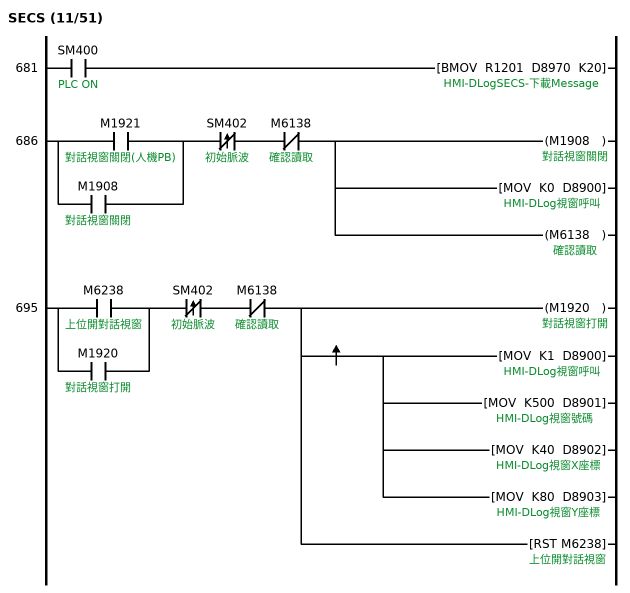
681   LD      SM400  ; PLC ON
      BMOV    R1201 D8970 K20  ; HMI-DLogSECS-下載Message
686   LD      M1921  ; 對話視窗關閉(人機PB)
      OR      M1908  ; 對話視窗關閉
      ANDPI   SM402  ; 初始脈波
      ANI     M6138  ; 確認讀取
      OUT     M1908  ; 對話視窗關閉
      MOV     K0 D8900  ; HMI-DLog視窗呼叫
      OUT     M6138  ; 確認讀取
695   LD      M6238  ; 上位開對話視窗
      OR      M1920  ; 對話視窗打開
      ANDPI   SM402  ; 初始脈波
      ANI     M6138  ; 確認讀取
      OUT     M1920  ; 對話視窗打開
      MPS
      MEP
      MOV     K1 D8900
      MOV     K500 D8901  ; HMI-DLog視窗號碼
      MOV     K40 D8902  ; HMI-DLog視窗X座標
      MOV     K80 D8903  ; HMI-DLog視窗Y座標
      MPP
      RST     M6238  ; 上位開對話視窗
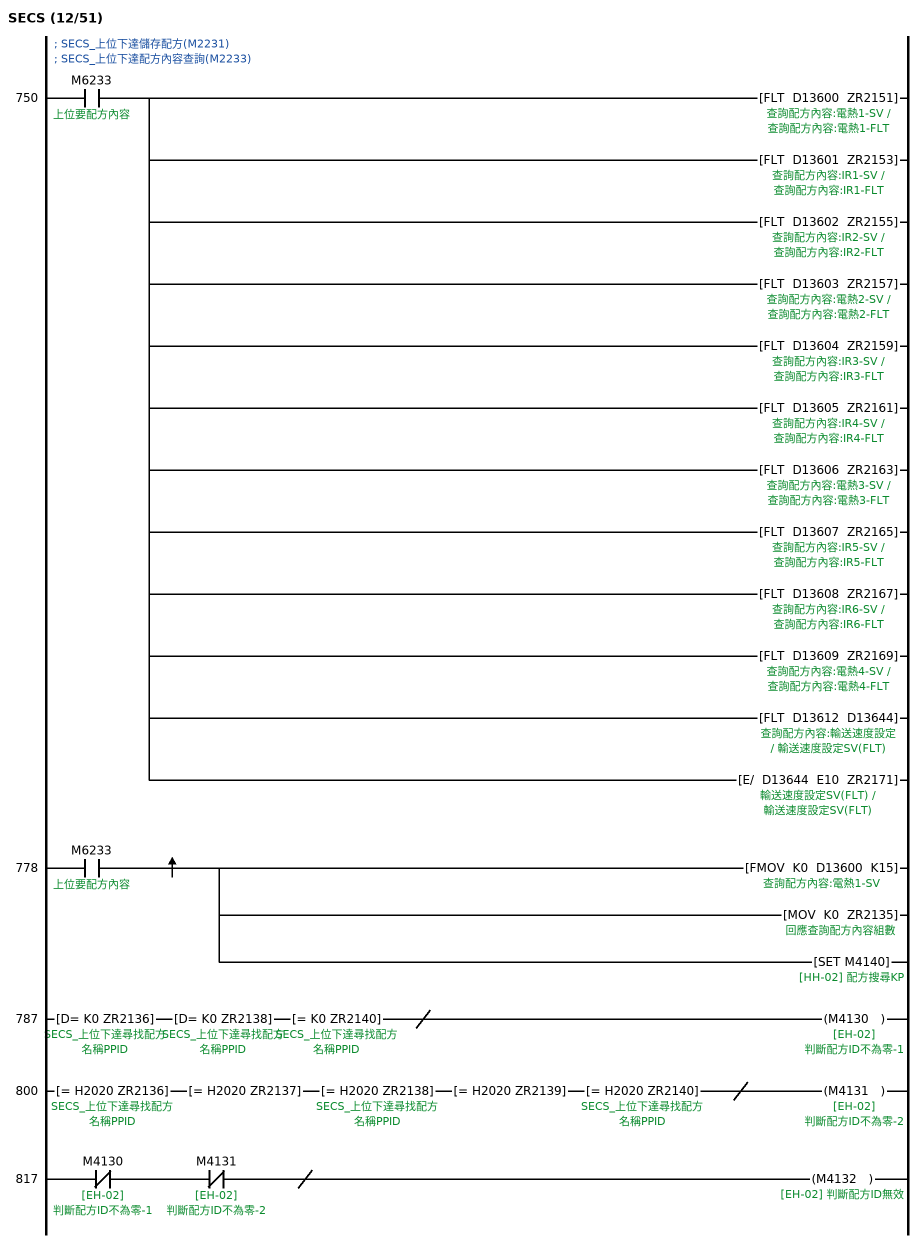
; SECS_上位下達儲存配方(M2231)
; SECS_上位下達配方內容查詢(M2233)
750   LD      M6233  ; 上位要配方內容
      FLT     D13600 ZR2151  ; 查詢配方內容:電熱1-SV / 查詢配方內容:電熱1-FLT
      FLT     D13601 ZR2153  ; 查詢配方內容:IR1-SV / 查詢配方內容:IR1-FLT
      FLT     D13602 ZR2155  ; 查詢配方內容:IR2-SV / 查詢配方內容:IR2-FLT
      FLT     D13603 ZR2157  ; 查詢配方內容:電熱2-SV / 查詢配方內容:電熱2-FLT
      FLT     D13604 ZR2159  ; 查詢配方內容:IR3-SV / 查詢配方內容:IR3-FLT
      FLT     D13605 ZR2161  ; 查詢配方內容:IR4-SV / 查詢配方內容:IR4-FLT
      FLT     D13606 ZR2163  ; 查詢配方內容:電熱3-SV / 查詢配方內容:電熱3-FLT
      FLT     D13607 ZR2165  ; 查詢配方內容:IR5-SV / 查詢配方內容:IR5-FLT
      FLT     D13608 ZR2167  ; 查詢配方內容:IR6-SV / 查詢配方內容:IR6-FLT
      FLT     D13609 ZR2169  ; 查詢配方內容:電熱4-SV / 查詢配方內容:電熱4-FLT
      FLT     D13612 D13644  ; 查詢配方內容:輸送速度設定 / 輸送速度設定SV(FLT)
      E/      D13644 E10 ZR2171  ; 輸送速度設定SV(FLT)
778   LD      M6233  ; 上位要配方內容
      MEP
      FMOV    K0 D13600 K15
      MOV     K0 ZR2135  ; 回應查詢配方內容組數
      SET     M4140  ; [HH-02] 配方搜尋KP
787   LDD=    K0 ZR2136  ; SECS_上位下達尋找配方名稱PPID
      ANDD=   K0 ZR2138  ; SECS_上位下達尋找配方名稱PPID
      AND=    K0 ZR2140  ; SECS_上位下達尋找配方名稱PPID
      INV
      OUT     M4130  ; [EH-02] 判斷配方ID不為零-1
800   LD=     H2020 ZR2136  ; SECS_上位下達尋找配方名稱PPID
      AND=    H2020 ZR2137
      AND=    H2020 ZR2138  ; SECS_上位下達尋找配方名稱PPID
      AND=    H2020 ZR2139
      AND=    H2020 ZR2140  ; SECS_上位下達尋找配方名稱PPID
      INV
      OUT     M4131  ; [EH-02] 判斷配方ID不為零-2
817   LDI     M4130  ; [EH-02] 判斷配方ID不為零-1
      ANI     M4131  ; [EH-02] 判斷配方ID不為零-2
      INV
      OUT     M4132  ; [EH-02] 判斷配方ID無效
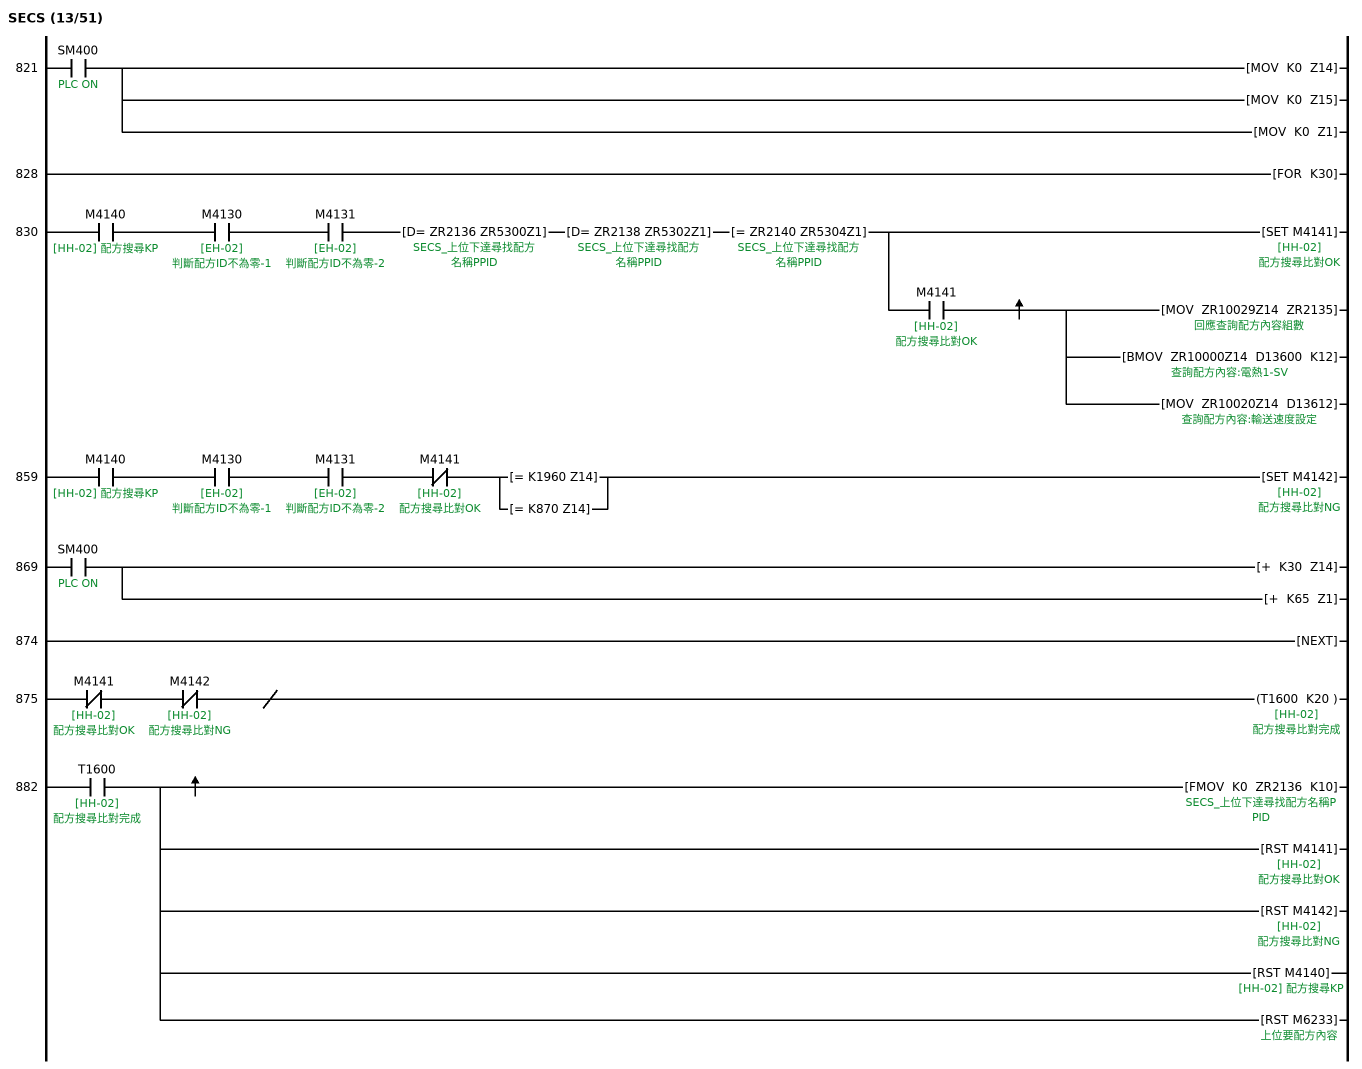
821   LD      SM400  ; PLC ON
      MOV     K0 Z14
      MOV     K0 Z15
      MOV     K0 Z1
828   FOR     K30
830   LD      M4140  ; [HH-02] 配方搜尋KP
      AND     M4130  ; [EH-02] 判斷配方ID不為零-1
      AND     M4131  ; [EH-02] 判斷配方ID不為零-2
      ANDD=   ZR2136 ZR5300Z1  ; SECS_上位下達尋找配方名稱PPID
      ANDD=   ZR2138 ZR5302Z1  ; SECS_上位下達尋找配方名稱PPID
      AND=    ZR2140 ZR5304Z1  ; SECS_上位下達尋找配方名稱PPID
      SET     M4141  ; [HH-02] 配方搜尋比對OK
      AND     M4141  ; [HH-02] 配方搜尋比對OK
      MEP
      MOV     ZR10029Z14 ZR2135
      BMOV    ZR10000Z14 D13600 K12
      MOV     ZR10020Z14 D13612
859   LD      M4140  ; [HH-02] 配方搜尋KP
      AND     M4130  ; [EH-02] 判斷配方ID不為零-1
      AND     M4131  ; [EH-02] 判斷配方ID不為零-2
      ANI     M4141  ; [HH-02] 配方搜尋比對OK
      LD=     K1960 Z14
      OR=     K870 Z14
      ANB
      SET     M4142  ; [HH-02] 配方搜尋比對NG
869   LD      SM400  ; PLC ON
      +       K30 Z14
      +       K65 Z1
874   NEXT
875   LDI     M4141  ; [HH-02] 配方搜尋比對OK
      ANI     M4142  ; [HH-02] 配方搜尋比對NG
      INV
      OUT     T1600 K20  ; [HH-02] 配方搜尋比對完成
882   LD      T1600  ; [HH-02] 配方搜尋比對完成
      MPS
      MEP
      FMOV    K0 ZR2136 K10
      MPP
      RST     M4141  ; [HH-02] 配方搜尋比對OK
      RST     M4142  ; [HH-02] 配方搜尋比對NG
      RST     M4140  ; [HH-02] 配方搜尋KP
      RST     M6233  ; 上位要配方內容
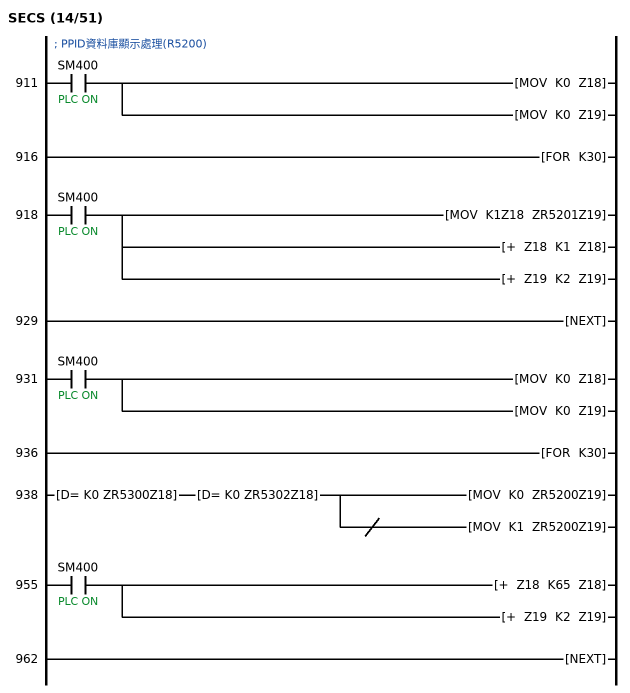
; PPID資料庫顯示處理(R5200)
911   LD      SM400  ; PLC ON
      MOV     K0 Z18
      MOV     K0 Z19
916   FOR     K30
918   LD      SM400  ; PLC ON
      MOV     K1Z18 ZR5201Z19
      +       Z18 K1 Z18
      +       Z19 K2 Z19
929   NEXT
931   LD      SM400  ; PLC ON
      MOV     K0 Z18
      MOV     K0 Z19
936   FOR     K30
938   LDD=    K0 ZR5300Z18
      ANDD=   K0 ZR5302Z18
      MOV     K0 ZR5200Z19
      INV
      MOV     K1 ZR5200Z19
955   LD      SM400  ; PLC ON
      +       Z18 K65 Z18
      +       Z19 K2 Z19
962   NEXT
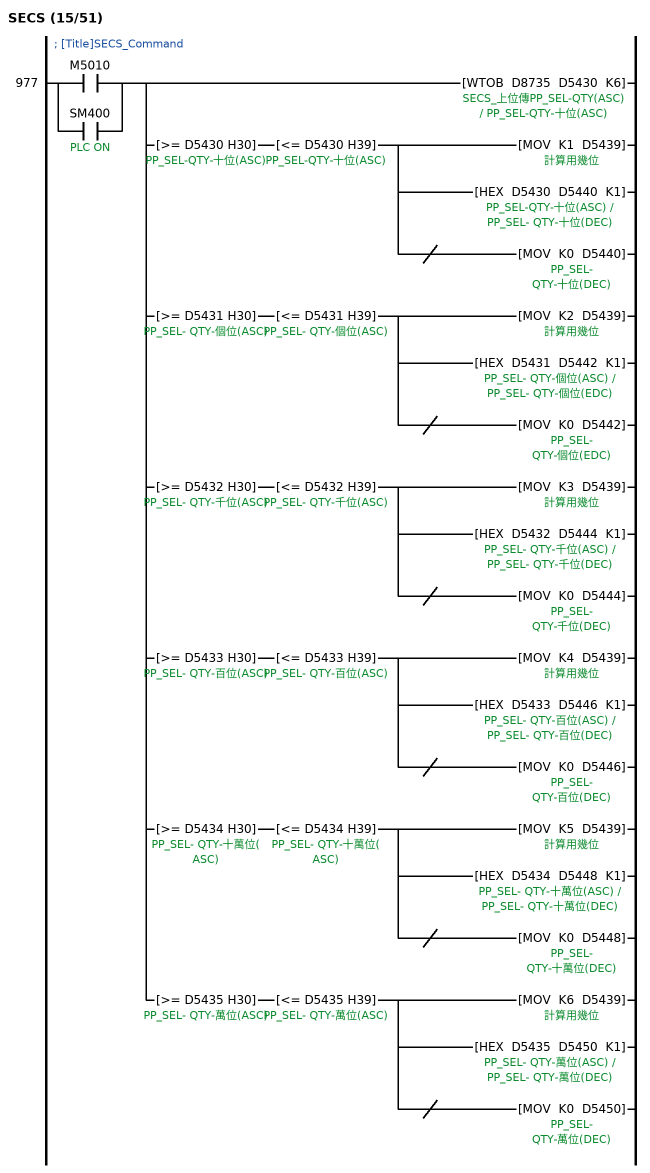
; [Title]SECS_Command
977   LD      M5010
      OR      SM400  ; PLC ON
      WTOB    D8735 D5430 K6  ; SECS_上位傳PP_SEL-QTY(ASC) / PP_SEL-QTY-十位(ASC)
      MPS
      AND>=   D5430 H30  ; PP_SEL-QTY-十位(ASC)
      AND<=   D5430 H39  ; PP_SEL-QTY-十位(ASC)
      MOV     K1 D5439  ; 計算用幾位
      HEX     D5430 D5440 K1  ; PP_SEL- QTY-十位(DEC)
      INV
      MOV     K0 D5440
      MRD
      AND>=   D5431 H30  ; PP_SEL- QTY-個位(ASC)
      AND<=   D5431 H39  ; PP_SEL- QTY-個位(ASC)
      MOV     K2 D5439
      HEX     D5431 D5442 K1  ; PP_SEL- QTY-個位(EDC)
      INV
      MOV     K0 D5442
      MRD
      AND>=   D5432 H30  ; PP_SEL- QTY-千位(ASC)
      AND<=   D5432 H39  ; PP_SEL- QTY-千位(ASC)
      MOV     K3 D5439
      HEX     D5432 D5444 K1  ; PP_SEL- QTY-千位(DEC)
      INV
      MOV     K0 D5444
      MRD
      AND>=   D5433 H30  ; PP_SEL- QTY-百位(ASC)
      AND<=   D5433 H39  ; PP_SEL- QTY-百位(ASC)
      MOV     K4 D5439
      HEX     D5433 D5446 K1  ; PP_SEL- QTY-百位(DEC)
      INV
      MOV     K0 D5446
      MRD
      AND>=   D5434 H30  ; PP_SEL- QTY-十萬位(ASC)
      AND<=   D5434 H39  ; PP_SEL- QTY-十萬位(ASC)
      MOV     K5 D5439
      HEX     D5434 D5448 K1  ; PP_SEL- QTY-十萬位(DEC)
      INV
      MOV     K0 D5448
      MPP
      AND>=   D5435 H30  ; PP_SEL- QTY-萬位(ASC)
      AND<=   D5435 H39  ; PP_SEL- QTY-萬位(ASC)
      MOV     K6 D5439
      HEX     D5435 D5450 K1  ; PP_SEL- QTY-萬位(DEC)
      INV
      MOV     K0 D5450
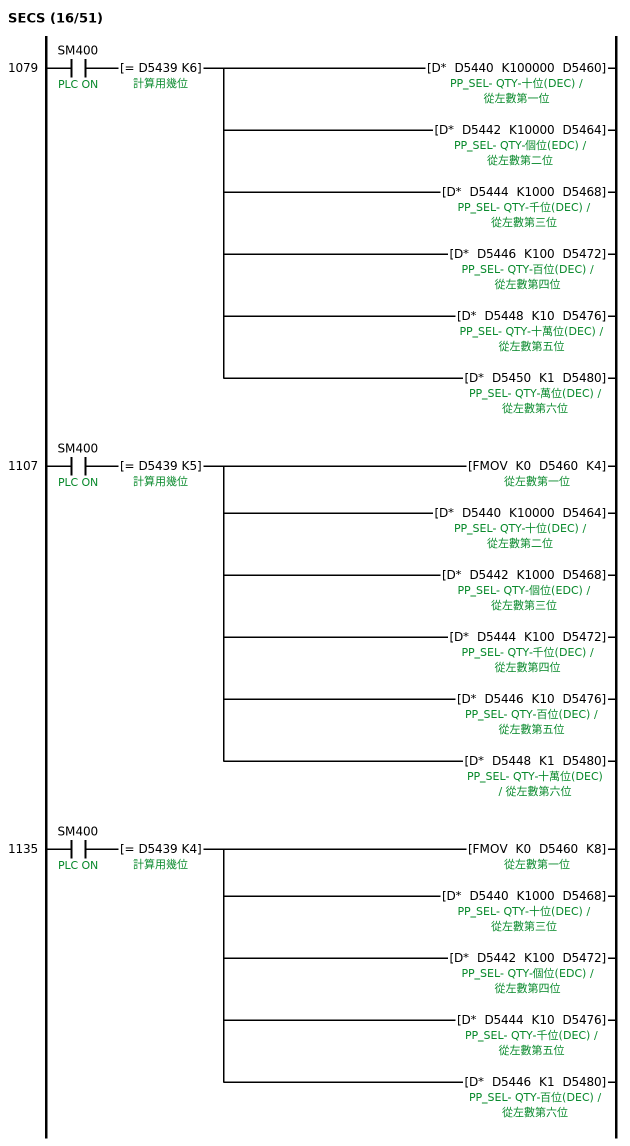
1079  LD      SM400  ; PLC ON
      AND=    D5439 K6  ; 計算用幾位
      D*      D5440 K100000 D5460  ; 從左數第一位
      D*      D5442 K10000 D5464  ; 從左數第二位
      D*      D5444 K1000 D5468  ; 從左數第三位
      D*      D5446 K100 D5472  ; 從左數第四位
      D*      D5448 K10 D5476  ; 從左數第五位
      D*      D5450 K1 D5480  ; 從左數第六位
1107  LD      SM400  ; PLC ON
      AND=    D5439 K5  ; 計算用幾位
      FMOV    K0 D5460 K4
      D*      D5440 K10000 D5464
      D*      D5442 K1000 D5468
      D*      D5444 K100 D5472
      D*      D5446 K10 D5476
      D*      D5448 K1 D5480
1135  LD      SM400  ; PLC ON
      AND=    D5439 K4  ; 計算用幾位
      FMOV    K0 D5460 K8
      D*      D5440 K1000 D5468
      D*      D5442 K100 D5472
      D*      D5444 K10 D5476
      D*      D5446 K1 D5480
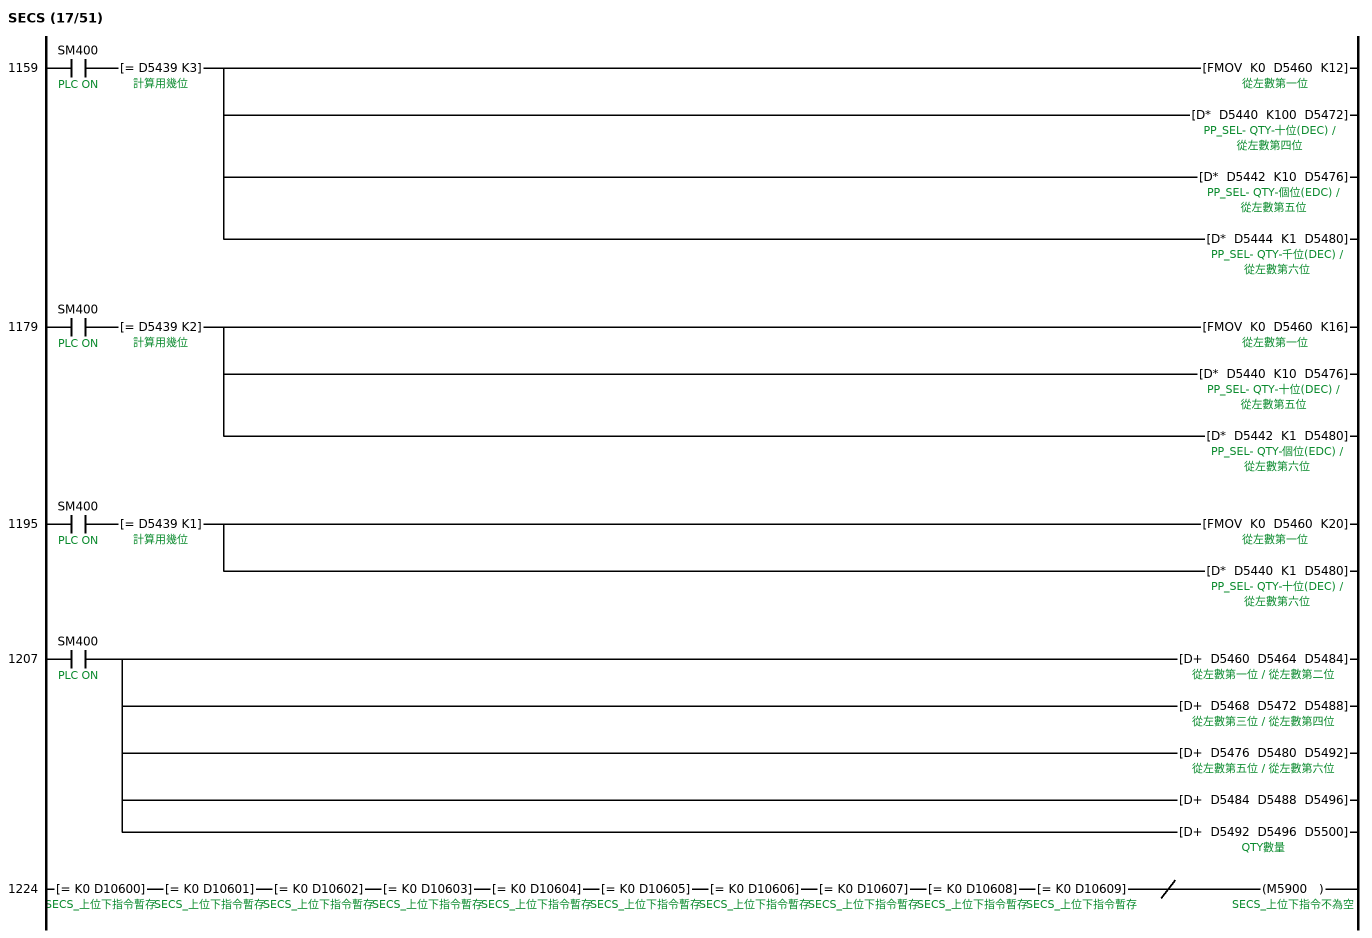
1159  LD      SM400  ; PLC ON
      AND=    D5439 K3  ; 計算用幾位
      FMOV    K0 D5460 K12
      D*      D5440 K100 D5472
      D*      D5442 K10 D5476
      D*      D5444 K1 D5480
1179  LD      SM400  ; PLC ON
      AND=    D5439 K2  ; 計算用幾位
      FMOV    K0 D5460 K16
      D*      D5440 K10 D5476
      D*      D5442 K1 D5480
1195  LD      SM400  ; PLC ON
      AND=    D5439 K1  ; 計算用幾位
      FMOV    K0 D5460 K20
      D*      D5440 K1 D5480
1207  LD      SM400  ; PLC ON
      D+      D5460 D5464 D5484
      D+      D5468 D5472 D5488
      D+      D5476 D5480 D5492
      D+      D5484 D5488 D5496
      D+      D5492 D5496 D5500  ; QTY數量
1224  LD=     K0 D10600  ; SECS_上位下指令暫存
      AND=    K0 D10601  ; SECS_上位下指令暫存
      AND=    K0 D10602  ; SECS_上位下指令暫存
      AND=    K0 D10603  ; SECS_上位下指令暫存
      AND=    K0 D10604  ; SECS_上位下指令暫存
      AND=    K0 D10605  ; SECS_上位下指令暫存
      AND=    K0 D10606  ; SECS_上位下指令暫存
      AND=    K0 D10607  ; SECS_上位下指令暫存
      AND=    K0 D10608  ; SECS_上位下指令暫存
      AND=    K0 D10609  ; SECS_上位下指令暫存
      INV
      OUT     M5900  ; SECS_上位下指令不為空
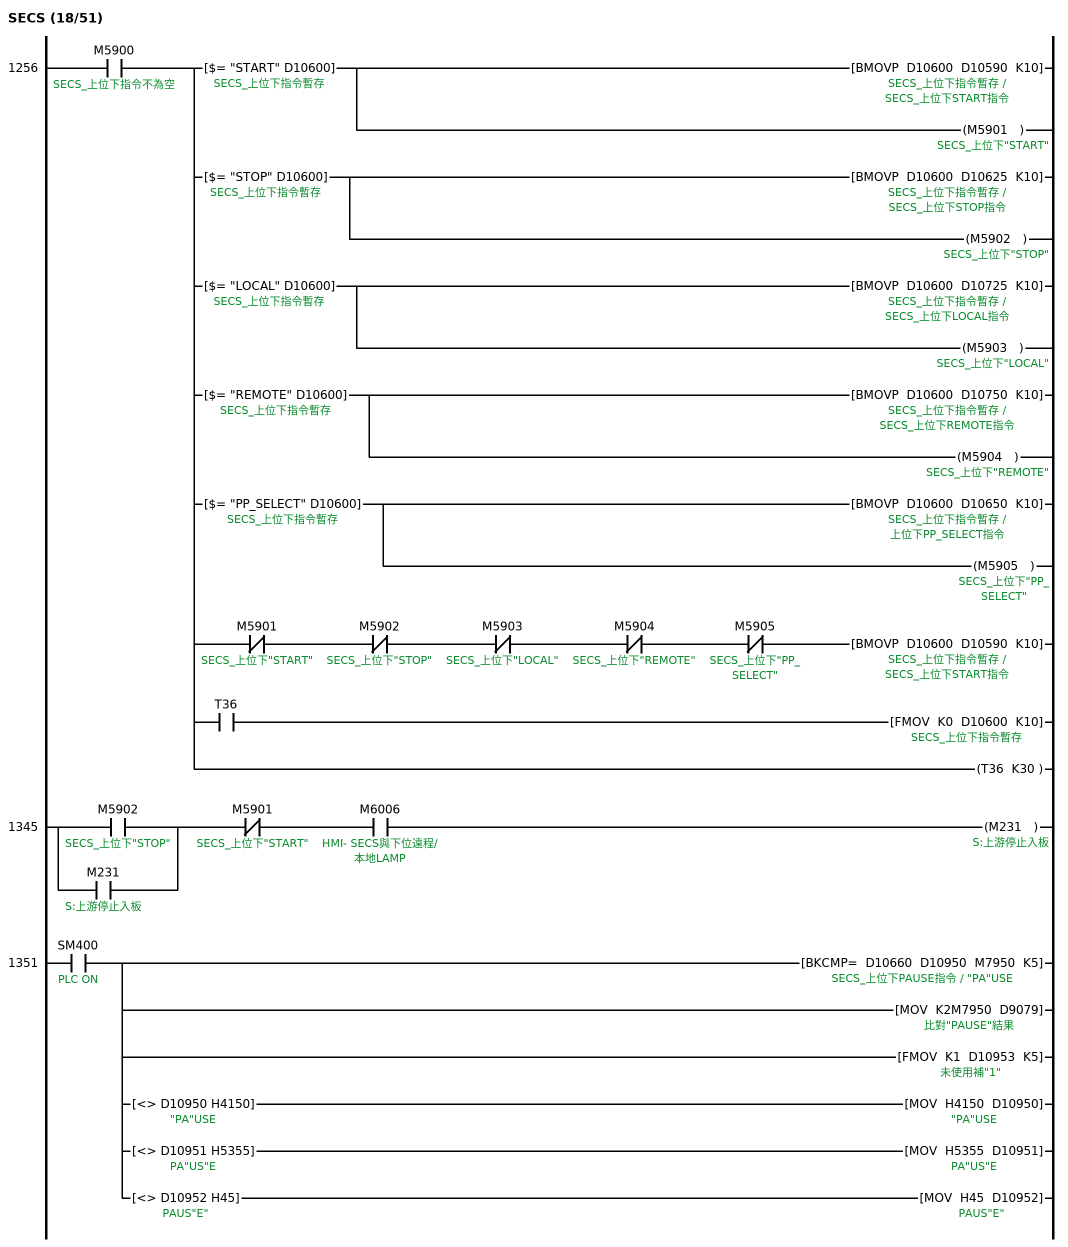
1256  LD      M5900  ; SECS_上位下指令不為空
      MPS
      AND$=   "START" D10600  ; SECS_上位下指令暫存
      BMOVP   D10600 D10590 K10  ; SECS_上位下START指令
      OUT     M5901  ; SECS_上位下"START"
      MRD
      AND$=   "STOP" D10600  ; SECS_上位下指令暫存
      BMOVP   D10600 D10625 K10  ; SECS_上位下STOP指令
      OUT     M5902  ; SECS_上位下"STOP"
      MRD
      AND$=   "LOCAL" D10600  ; SECS_上位下指令暫存
      BMOVP   D10600 D10725 K10  ; SECS_上位下LOCAL指令
      OUT     M5903  ; SECS_上位下"LOCAL"
      MRD
      AND$=   "REMOTE" D10600  ; SECS_上位下指令暫存
      BMOVP   D10600 D10750 K10  ; SECS_上位下REMOTE指令
      OUT     M5904  ; SECS_上位下"REMOTE"
      MRD
      AND$=   "PP_SELECT" D10600  ; SECS_上位下指令暫存
      BMOVP   D10600 D10650 K10  ; 上位下PP_SELECT指令
      OUT     M5905  ; SECS_上位下"PP_SELECT"
      MRD
      ANI     M5901  ; SECS_上位下"START"
      ANI     M5902  ; SECS_上位下"STOP"
      ANI     M5903  ; SECS_上位下"LOCAL"
      ANI     M5904  ; SECS_上位下"REMOTE"
      ANI     M5905  ; SECS_上位下"PP_SELECT"
      BMOVP   D10600 D10590 K10
      MRD
      AND     T36
      FMOV    K0 D10600 K10
      MPP
      OUT     T36 K30
1345  LD      M5902  ; SECS_上位下"STOP"
      OR      M231  ; S:上游停止入板
      ANI     M5901  ; SECS_上位下"START"
      AND     M6006  ; HMI- SECS與下位遠程/本地LAMP
      OUT     M231  ; S:上游停止入板
1351  LD      SM400  ; PLC ON
      BKCMP=  D10660 D10950 M7950 K5  ; SECS_上位下PAUSE指令 / "PA"USE
        [note] 上位下PAUSE指令
      MOV     K2M7950 D9079  ; 比對"PAUSE"結果
      FMOV    K1 D10953 K5  ; 未使用補"1"
      MPS
      AND<>   D10950 H4150  ; "PA"USE
      MOV     H4150 D10950
      MRD
      AND<>   D10951 H5355  ; PA"US"E
      MOV     H5355 D10951
      MPP
      AND<>   D10952 H45  ; PAUS"E"
      MOV     H45 D10952
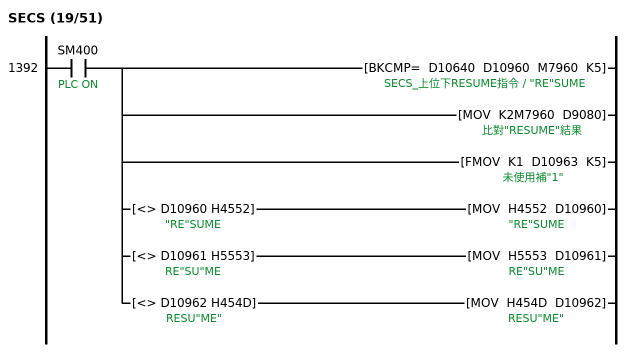
1392  LD      SM400  ; PLC ON
      BKCMP=  D10640 D10960 M7960 K5  ; SECS_上位下RESUME指令 / "RE"SUME
        [note] 上位下RESUME指令
      MOV     K2M7960 D9080  ; 比對"RESUME"結果
      FMOV    K1 D10963 K5  ; 未使用補"1"
      MPS
      AND<>   D10960 H4552  ; "RE"SUME
      MOV     H4552 D10960
      MRD
      AND<>   D10961 H5553  ; RE"SU"ME
      MOV     H5553 D10961
      MPP
      AND<>   D10962 H454D  ; RESU"ME"
      MOV     H454D D10962
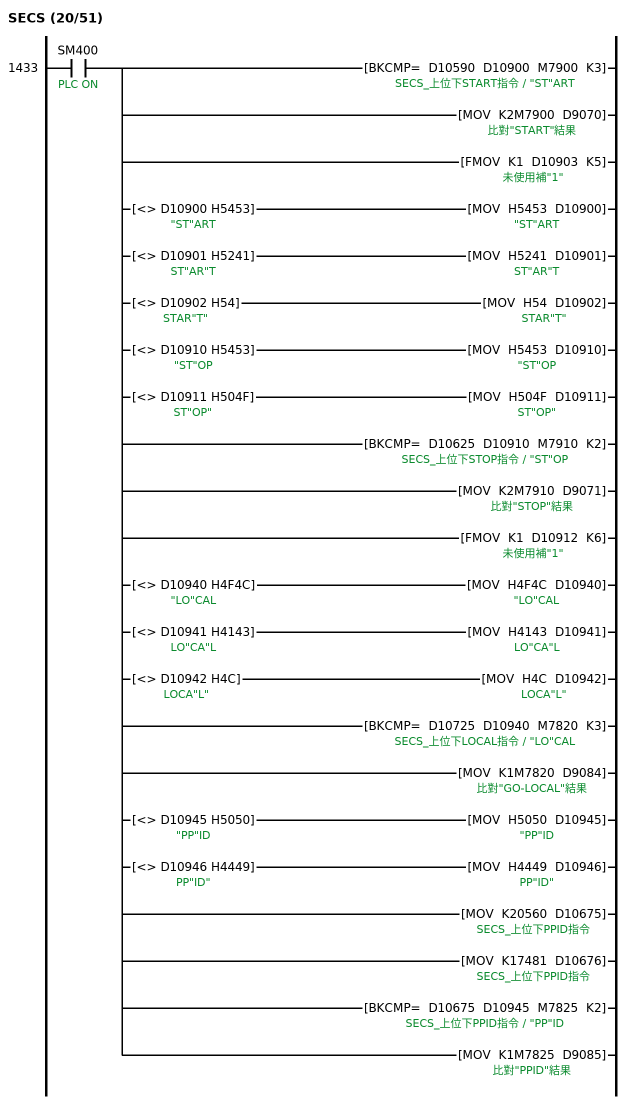
1433  LD      SM400  ; PLC ON
      BKCMP=  D10590 D10900 M7900 K3  ; "ST"ART
        [note] 上位下START指令
      MOV     K2M7900 D9070  ; 比對"START"結果
      FMOV    K1 D10903 K5  ; 未使用補"1"
      MPS
      AND<>   D10900 H5453  ; "ST"ART
      MOV     H5453 D10900
      MRD
      AND<>   D10901 H5241  ; ST"AR"T
      MOV     H5241 D10901
      MRD
      AND<>   D10902 H54  ; STAR"T"
      MOV     H54 D10902
      MRD
      AND<>   D10910 H5453  ; "ST"OP
      MOV     H5453 D10910
      MRD
      AND<>   D10911 H504F  ; ST"OP"
      MOV     H504F D10911
      MPP
      BKCMP=  D10625 D10910 M7910 K2
        [note] 上位下STOP指令
      MOV     K2M7910 D9071  ; 比對"STOP"結果
      FMOV    K1 D10912 K6  ; 未使用補"1"
      MPS
      AND<>   D10940 H4F4C  ; "LO"CAL
      MOV     H4F4C D10940
      MRD
      AND<>   D10941 H4143  ; LO"CA"L
      MOV     H4143 D10941
      MRD
      AND<>   D10942 H4C  ; LOCA"L"
      MOV     H4C D10942
      MPP
      BKCMP=  D10725 D10940 M7820 K3
        [note] 上位下GO-LOCAL指令
      MOV     K1M7820 D9084  ; 比對"GO-LOCAL"結果
      MPS
      AND<>   D10945 H5050  ; "PP"ID
      MOV     H5050 D10945
      MRD
      AND<>   D10946 H4449  ; PP"ID"
      MOV     H4449 D10946
      MPP
      MOV     K20560 D10675  ; SECS_上位下PPID指令
      MOV     K17481 D10676  ; SECS_上位下PPID指令
      BKCMP=  D10675 D10945 M7825 K2
        [note] 上位下PPID指令
      MOV     K1M7825 D9085  ; 比對"PPID"結果
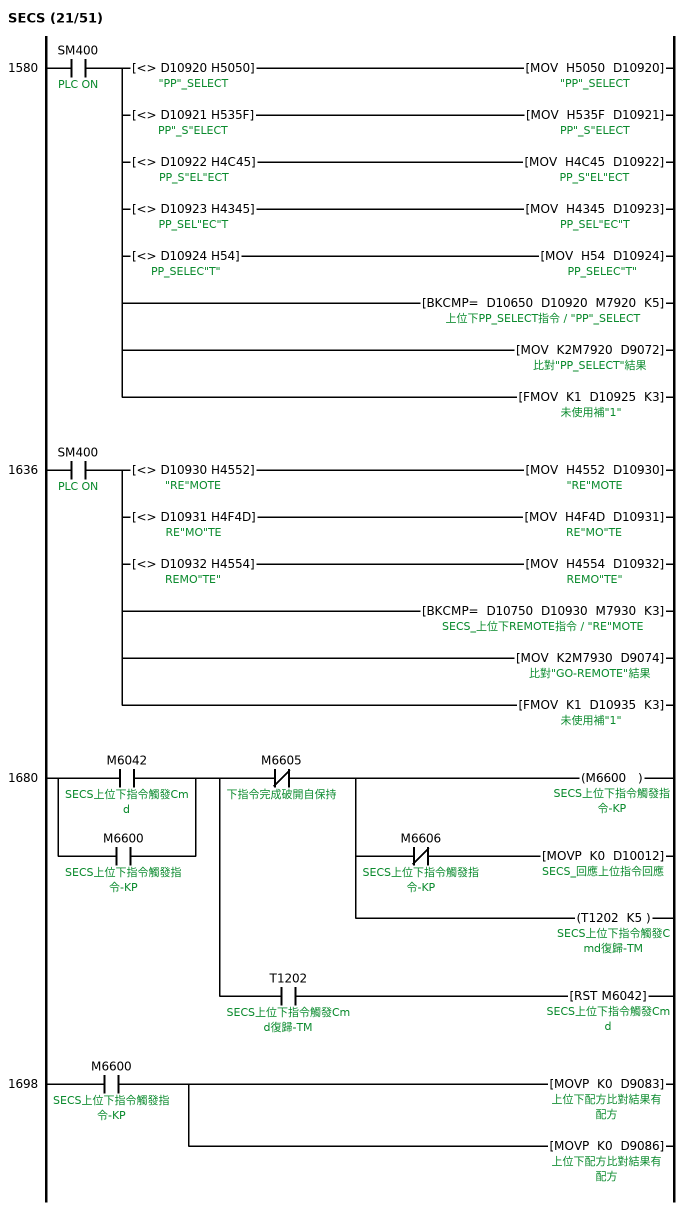
1580  LD      SM400  ; PLC ON
      MPS
      AND<>   D10920 H5050  ; "PP"_SELECT
      MOV     H5050 D10920
      MRD
      AND<>   D10921 H535F  ; PP"_S"ELECT
      MOV     H535F D10921
      MRD
      AND<>   D10922 H4C45  ; PP_S"EL"ECT
      MOV     H4C45 D10922
      MRD
      AND<>   D10923 H4345  ; PP_SEL"EC"T
      MOV     H4345 D10923
      MRD
      AND<>   D10924 H54  ; PP_SELEC"T"
      MOV     H54 D10924
      MPP
      BKCMP=  D10650 D10920 M7920 K5
        [note] 上位下PP_SELECT指令
      MOV     K2M7920 D9072  ; 比對"PP_SELECT"結果
      FMOV    K1 D10925 K3  ; 未使用補"1"
1636  LD      SM400  ; PLC ON
      MPS
      AND<>   D10930 H4552  ; "RE"MOTE
      MOV     H4552 D10930
      MRD
      AND<>   D10931 H4F4D  ; RE"MO"TE
      MOV     H4F4D D10931
      MRD
      AND<>   D10932 H4554  ; REMO"TE"
      MOV     H4554 D10932
      MPP
      BKCMP=  D10750 D10930 M7930 K3
        [note] 上位下GO-REMOTE指令
      MOV     K2M7930 D9074  ; 比對"GO-REMOTE"結果
      FMOV    K1 D10935 K3  ; 未使用補"1"
1680  LD      M6042  ; SECS上位下指令觸發Cmd
      OR      M6600  ; SECS上位下指令觸發指令-KP
      MPS
      ANI     M6605  ; 下指令完成破開自保持
      OUT     M6600  ; SECS上位下指令觸發指令-KP
      MPS
      ANI     M6606  ; SECS上位下指令觸發指令-KP
      MOVP    K0 D10012  ; SECS_回應上位指令回應
      MPP
      OUT     T1202 K5  ; SECS上位下指令觸發Cmd復歸-TM
      MPP
      AND     T1202  ; SECS上位下指令觸發Cmd復歸-TM
      RST     M6042  ; SECS上位下指令觸發Cmd
1698  LD      M6600  ; SECS上位下指令觸發指令-KP
      MOVP    K0 D9083  ; 上位下配方比對結果有配方
      MOVP    K0 D9086  ; 上位下配方比對結果有配方
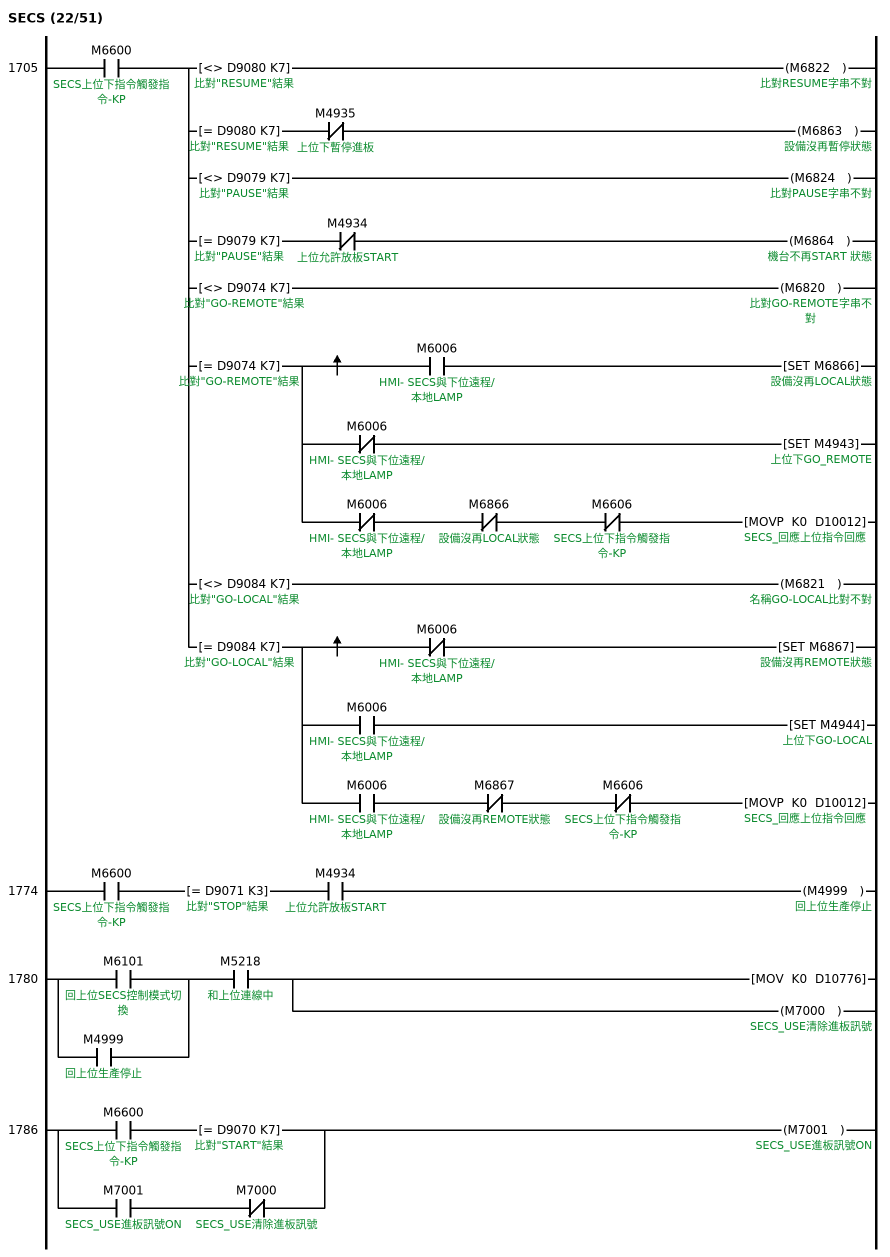
1705  LD      M6600  ; SECS上位下指令觸發指令-KP
      MPS
      AND<>   D9080 K7  ; 比對"RESUME"結果
      OUT     M6822  ; 比對RESUME字串不對
      MRD
      AND=    D9080 K7  ; 比對"RESUME"結果
      ANI     M4935  ; 上位下暫停進板
      OUT     M6863  ; 設備沒再暫停狀態
      MRD
      AND<>   D9079 K7  ; 比對"PAUSE"結果
      OUT     M6824  ; 比對PAUSE字串不對
      MRD
      AND=    D9079 K7  ; 比對"PAUSE"結果
      ANI     M4934  ; 上位允許放板START
      OUT     M6864  ; 機台不再START 狀態
      MRD
      AND<>   D9074 K7  ; 比對"GO-REMOTE"結果
      OUT     M6820  ; 比對GO-REMOTE字串不對
      MRD
      AND=    D9074 K7  ; 比對"GO-REMOTE"結果
      MPS
      MEP
      AND     M6006  ; HMI- SECS與下位遠程/本地LAMP
      SET     M6866  ; 設備沒再LOCAL狀態
      MRD
      ANI     M6006  ; HMI- SECS與下位遠程/本地LAMP
      SET     M4943  ; 上位下GO_REMOTE
      MPP
      ANI     M6006  ; HMI- SECS與下位遠程/本地LAMP
      ANI     M6866  ; 設備沒再LOCAL狀態
      ANI     M6606  ; SECS上位下指令觸發指令-KP
      MOVP    K0 D10012
      MRD
      AND<>   D9084 K7  ; 比對"GO-LOCAL"結果
      OUT     M6821  ; 名稱GO-LOCAL比對不對
      MPP
      AND=    D9084 K7  ; 比對"GO-LOCAL"結果
      MPS
      MEP
      ANI     M6006  ; HMI- SECS與下位遠程/本地LAMP
      SET     M6867  ; 設備沒再REMOTE狀態
      MRD
      AND     M6006  ; HMI- SECS與下位遠程/本地LAMP
      SET     M4944  ; 上位下GO-LOCAL
      MPP
      AND     M6006  ; HMI- SECS與下位遠程/本地LAMP
      ANI     M6867  ; 設備沒再REMOTE狀態
      ANI     M6606  ; SECS上位下指令觸發指令-KP
      MOVP    K0 D10012
1774  LD      M6600  ; SECS上位下指令觸發指令-KP
      AND=    D9071 K3  ; 比對"STOP"結果
      AND     M4934  ; 上位允許放板START
      OUT     M4999  ; 回上位生產停止
1780  LD      M6101  ; 回上位SECS控制模式切換
      OR      M4999  ; 回上位生產停止
      AND     M5218  ; 和上位連線中
      MOV     K0 D10776
      OUT     M7000  ; SECS_USE清除進板訊號
1786  LD      M6600  ; SECS上位下指令觸發指令-KP
      AND=    D9070 K7  ; 比對"START"結果
      LD      M7001  ; SECS_USE進板訊號ON
      ANI     M7000  ; SECS_USE清除進板訊號
      ORB
      OUT     M7001  ; SECS_USE進板訊號ON
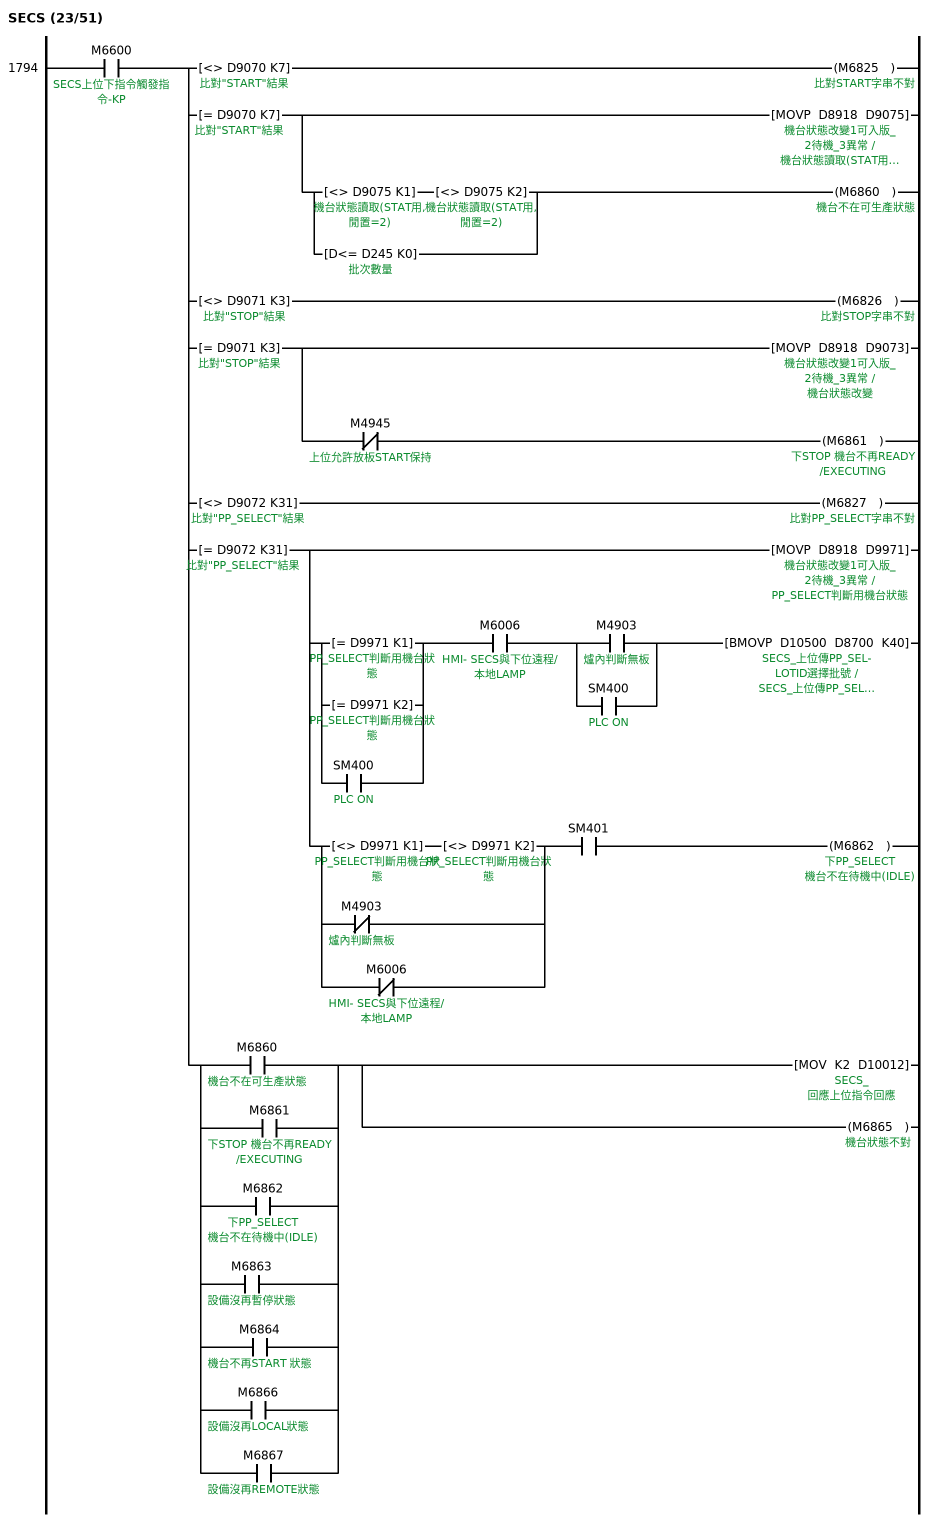
1794  LD      M6600  ; SECS上位下指令觸發指令-KP
      MPS
      AND<>   D9070 K7  ; 比對"START"結果
      OUT     M6825  ; 比對START字串不對
      MRD
      AND=    D9070 K7  ; 比對"START"結果
      MOVP    D8918 D9075  ; 機台狀態讀取(STAT用,閒置=2)
      LD<>    D9075 K1  ; 機台狀態讀取(STAT用,閒置=2)
      AND<>   D9075 K2  ; 機台狀態讀取(STAT用,閒置=2)
      ORD<=   D245 K0  ; 批次數量
      ANB
      OUT     M6860  ; 機台不在可生產狀態
      MRD
      AND<>   D9071 K3  ; 比對"STOP"結果
      OUT     M6826  ; 比對STOP字串不對
      MRD
      AND=    D9071 K3  ; 比對"STOP"結果
      MOVP    D8918 D9073  ; 機台狀態改變
      ANI     M4945  ; 上位允許放板START保持
      OUT     M6861  ; 下STOP 機台不再READY/EXECUTING
      MRD
      AND<>   D9072 K31  ; 比對"PP_SELECT"結果
      OUT     M6827  ; 比對PP_SELECT字串不對
      MRD
      AND=    D9072 K31  ; 比對"PP_SELECT"結果
      MOVP    D8918 D9971  ; PP_SELECT判斷用機台狀態
      MPS
      LD=     D9971 K1  ; PP_SELECT判斷用機台狀態
      OR=     D9971 K2  ; PP_SELECT判斷用機台狀態
      OR      SM400  ; PLC ON
      ANB
      AND     M6006  ; HMI- SECS與下位遠程/本地LAMP
      LD      M4903  ; 爐內判斷無板
      OR      SM400  ; PLC ON
      ANB
      BMOVP   D10500 D8700 K40  ; SECS_上位傳PP_SEL-LOTID選擇批號 / SECS_上位傳PP_SEL-LOTID選擇批號
      MPP
      LD<>    D9971 K1  ; PP_SELECT判斷用機台狀態
      AND<>   D9971 K2  ; PP_SELECT判斷用機台狀態
      ORI     M4903  ; 爐內判斷無板
      ORI     M6006  ; HMI- SECS與下位遠程/本地LAMP
      ANB
      AND     SM401
      OUT     M6862  ; 下PP_SELECT 機台不在待機中(IDLE)
      MPP
      LD      M6860  ; 機台不在可生產狀態
      OR      M6861  ; 下STOP 機台不再READY/EXECUTING
      OR      M6862  ; 下PP_SELECT 機台不在待機中(IDLE)
      OR      M6863  ; 設備沒再暫停狀態
      OR      M6864  ; 機台不再START 狀態
      OR      M6866  ; 設備沒再LOCAL狀態
      OR      M6867  ; 設備沒再REMOTE狀態
      ANB
      MOV     K2 D10012
      OUT     M6865  ; 機台狀態不對
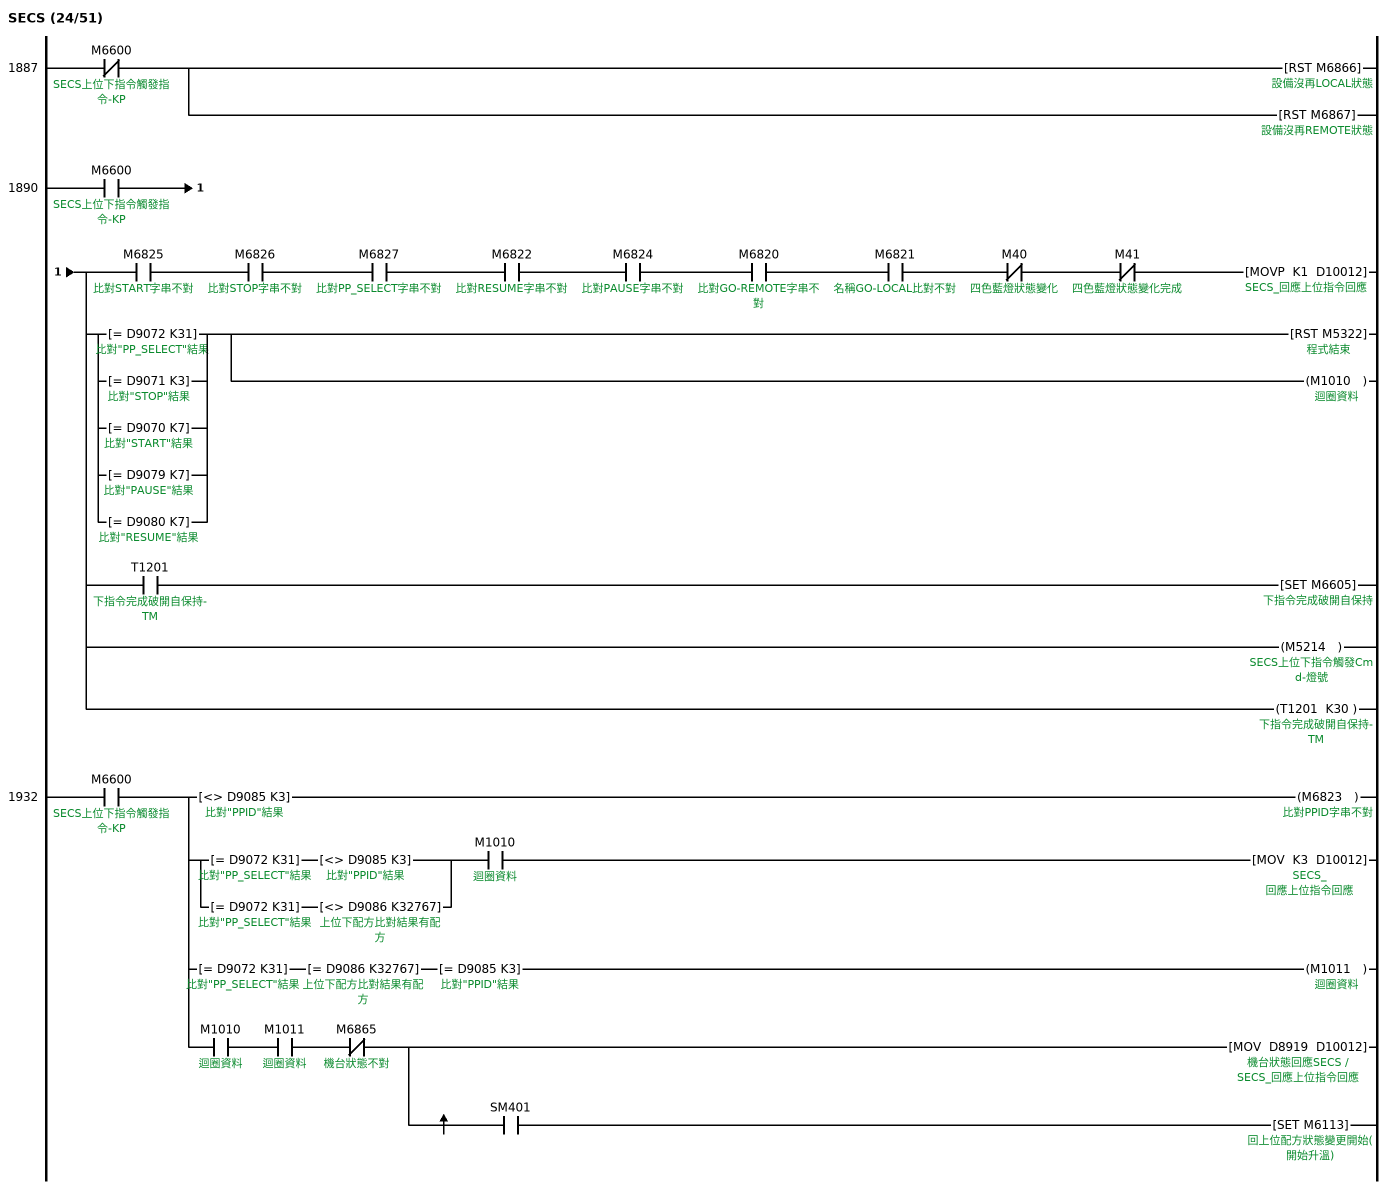
1887  LDI     M6600  ; SECS上位下指令觸發指令-KP
      RST     M6866  ; 設備沒再LOCAL狀態
      RST     M6867  ; 設備沒再REMOTE狀態
1890  LD      M6600  ; SECS上位下指令觸發指令-KP
      MPS
      AND     M6825  ; 比對START字串不對
      AND     M6826  ; 比對STOP字串不對
      AND     M6827  ; 比對PP_SELECT字串不對
      AND     M6822  ; 比對RESUME字串不對
      AND     M6824  ; 比對PAUSE字串不對
      AND     M6820  ; 比對GO-REMOTE字串不對
      AND     M6821  ; 名稱GO-LOCAL比對不對
      ANI     M40  ; 四色藍燈狀態變化
      ANI     M41  ; 四色藍燈狀態變化完成
      MOVP    K1 D10012
      MRD
      LD=     D9072 K31  ; 比對"PP_SELECT"結果
      OR=     D9071 K3  ; 比對"STOP"結果
      OR=     D9070 K7  ; 比對"START"結果
      OR=     D9079 K7  ; 比對"PAUSE"結果
      OR=     D9080 K7  ; 比對"RESUME"結果
      ANB
      RST     M5322  ; 程式結束
      OUT     M1010  ; 迴圈資料
      MRD
      AND     T1201  ; 下指令完成破開自保持-TM
      SET     M6605  ; 下指令完成破開自保持
      MPP
      OUT     M5214  ; SECS上位下指令觸發Cmd-燈號
      OUT     T1201 K30  ; 下指令完成破開自保持-TM
1932  LD      M6600  ; SECS上位下指令觸發指令-KP
      MPS
      AND<>   D9085 K3  ; 比對"PPID"結果
      OUT     M6823  ; 比對PPID字串不對
      MRD
      LD=     D9072 K31  ; 比對"PP_SELECT"結果
      AND<>   D9085 K3  ; 比對"PPID"結果
      LD=     D9072 K31  ; 比對"PP_SELECT"結果
      AND<>   D9086 K32767  ; 上位下配方比對結果有配方
      ORB
      ANB
      AND     M1010  ; 迴圈資料
      MOV     K3 D10012
      MRD
      AND=    D9072 K31  ; 比對"PP_SELECT"結果
      AND=    D9086 K32767  ; 上位下配方比對結果有配方
      AND=    D9085 K3  ; 比對"PPID"結果
      OUT     M1011  ; 迴圈資料
      MPP
      AND     M1010  ; 迴圈資料
      AND     M1011  ; 迴圈資料
      ANI     M6865  ; 機台狀態不對
      MOV     D8919 D10012  ; 機台狀態回應SECS
      MEP
      AND     SM401
      SET     M6113  ; 回上位配方狀態變更開始(開始升溫)
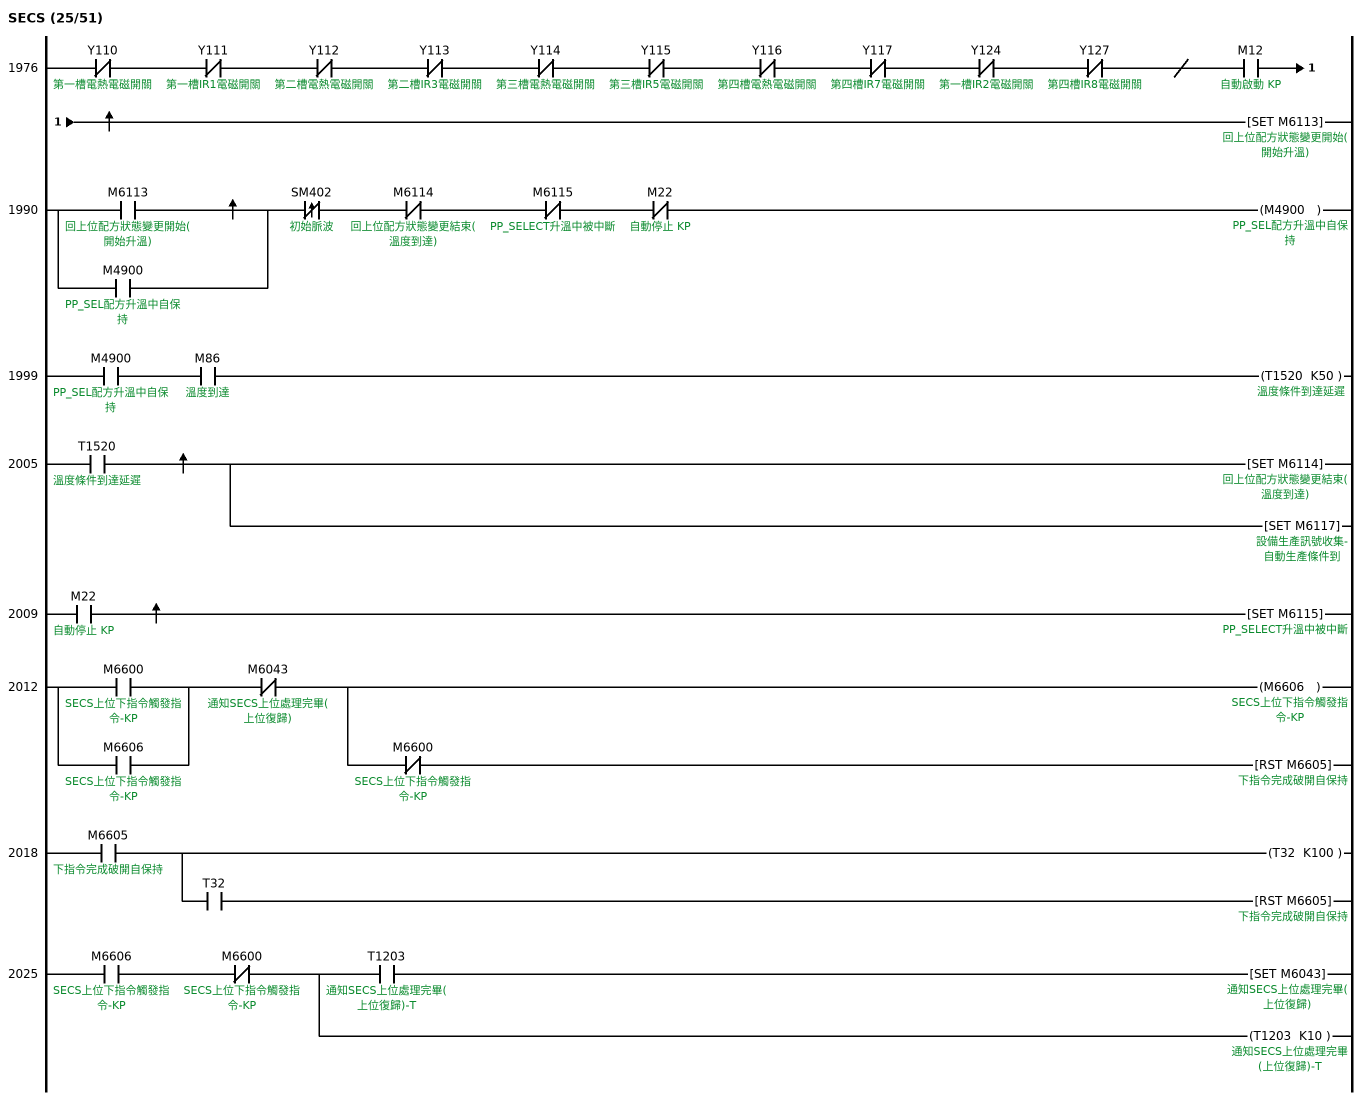
1976  LDI     Y110  ; 第一槽電熱電磁開關
      ANI     Y111  ; 第一槽IR1電磁開關
      ANI     Y112  ; 第二槽電熱電磁開關
      ANI     Y113  ; 第二槽IR3電磁開關
      ANI     Y114  ; 第三槽電熱電磁開關
      ANI     Y115  ; 第三槽IR5電磁開關
      ANI     Y116  ; 第四槽電熱電磁開關
      ANI     Y117  ; 第四槽IR7電磁開關
      ANI     Y124  ; 第一槽IR2電磁開關
      ANI     Y127  ; 第四槽IR8電磁開關
      INV
      AND     M12  ; 自動啟動 KP
      MEP
      SET     M6113  ; 回上位配方狀態變更開始(開始升溫)
1990  LD      M6113  ; 回上位配方狀態變更開始(開始升溫)
      MEP
      OR      M4900  ; PP_SEL配方升溫中自保持
      ANDPI   SM402  ; 初始脈波
      ANI     M6114  ; 回上位配方狀態變更結束(溫度到達)
      ANI     M6115  ; PP_SELECT升溫中被中斷
      ANI     M22  ; 自動停止 KP
      OUT     M4900  ; PP_SEL配方升溫中自保持
1999  LD      M4900  ; PP_SEL配方升溫中自保持
      AND     M86  ; 溫度到達
      OUT     T1520 K50  ; 溫度條件到達延遲
2005  LD      T1520  ; 溫度條件到達延遲
      MEP
      SET     M6114  ; 回上位配方狀態變更結束(溫度到達)
      SET     M6117  ; 設備生產訊號收集-自動生產條件到
2009  LD      M22  ; 自動停止 KP
      MEP
      SET     M6115  ; PP_SELECT升溫中被中斷
2012  LD      M6600  ; SECS上位下指令觸發指令-KP
      OR      M6606  ; SECS上位下指令觸發指令-KP
      ANI     M6043  ; 通知SECS上位處理完畢(上位復歸)
      OUT     M6606  ; SECS上位下指令觸發指令-KP
      ANI     M6600  ; SECS上位下指令觸發指令-KP
      RST     M6605  ; 下指令完成破開自保持
2018  LD      M6605  ; 下指令完成破開自保持
      OUT     T32 K100
      AND     T32
      RST     M6605  ; 下指令完成破開自保持
2025  LD      M6606  ; SECS上位下指令觸發指令-KP
      ANI     M6600  ; SECS上位下指令觸發指令-KP
      MPS
      AND     T1203  ; 通知SECS上位處理完畢(上位復歸)-T
      SET     M6043  ; 通知SECS上位處理完畢(上位復歸)
      MPP
      OUT     T1203 K10  ; 通知SECS上位處理完畢(上位復歸)-T
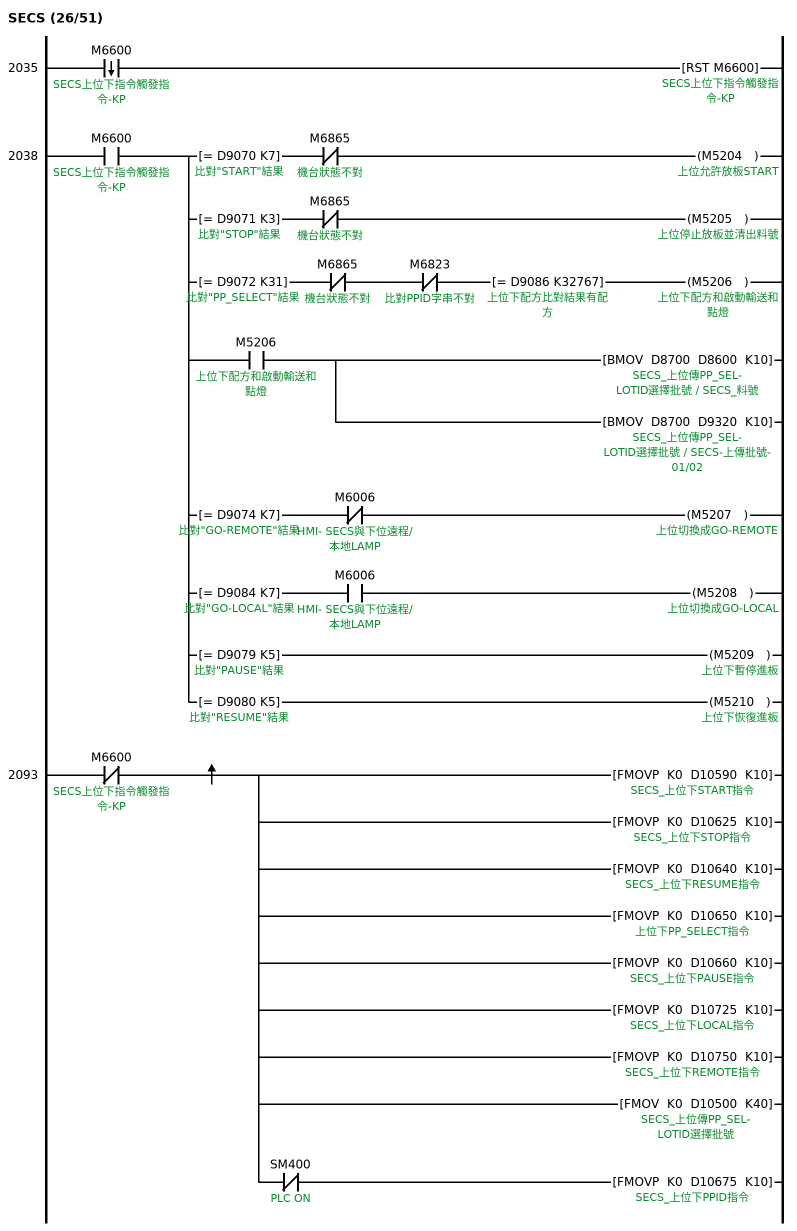
2035  LDF     M6600  ; SECS上位下指令觸發指令-KP
      RST     M6600  ; SECS上位下指令觸發指令-KP
2038  LD      M6600  ; SECS上位下指令觸發指令-KP
      MPS
      AND=    D9070 K7  ; 比對"START"結果
      ANI     M6865  ; 機台狀態不對
      OUT     M5204  ; 上位允許放板START
      MRD
      AND=    D9071 K3  ; 比對"STOP"結果
      ANI     M6865  ; 機台狀態不對
      OUT     M5205  ; 上位停止放板並清出料號
      MRD
      AND=    D9072 K31  ; 比對"PP_SELECT"結果
      ANI     M6865  ; 機台狀態不對
      ANI     M6823  ; 比對PPID字串不對
      AND=    D9086 K32767  ; 上位下配方比對結果有配方
      OUT     M5206  ; 上位下配方和啟動輸送和點燈
      MRD
      AND     M5206  ; 上位下配方和啟動輸送和點燈
      BMOV    D8700 D8600 K10  ; SECS_料號
      BMOV    D8700 D9320 K10  ; SECS-上傳批號-   01/02
      MRD
      AND=    D9074 K7  ; 比對"GO-REMOTE"結果
      ANI     M6006  ; HMI- SECS與下位遠程/本地LAMP
      OUT     M5207  ; 上位切換成GO-REMOTE
      MRD
      AND=    D9084 K7  ; 比對"GO-LOCAL"結果
      AND     M6006  ; HMI- SECS與下位遠程/本地LAMP
      OUT     M5208  ; 上位切換成GO-LOCAL
      MRD
      AND=    D9079 K5  ; 比對"PAUSE"結果
      OUT     M5209  ; 上位下暫停進板
      MPP
      AND=    D9080 K5  ; 比對"RESUME"結果
      OUT     M5210  ; 上位下恢復進板
2093  LDI     M6600  ; SECS上位下指令觸發指令-KP
      MEP
      FMOVP   K0 D10590 K10
      FMOVP   K0 D10625 K10
      FMOVP   K0 D10640 K10
      FMOVP   K0 D10650 K10
      FMOVP   K0 D10660 K10
      FMOVP   K0 D10725 K10
      FMOVP   K0 D10750 K10
      FMOV    K0 D10500 K40
      ANI     SM400  ; PLC ON
      FMOVP   K0 D10675 K10
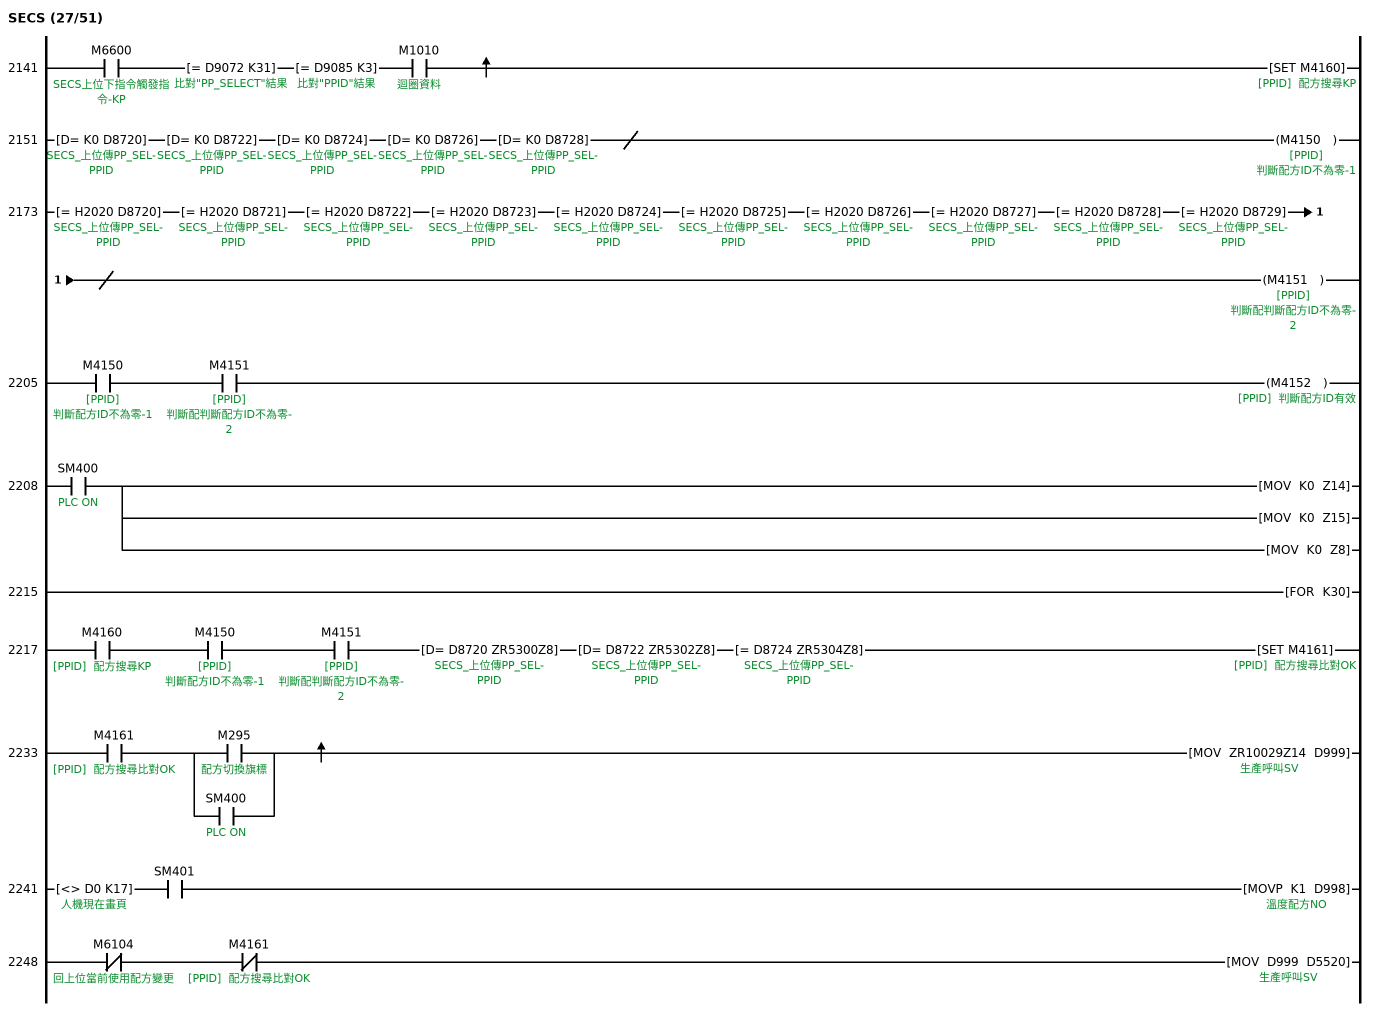
2141  LD      M6600  ; SECS上位下指令觸發指令-KP
      AND=    D9072 K31  ; 比對"PP_SELECT"結果
      AND=    D9085 K3  ; 比對"PPID"結果
      AND     M1010  ; 迴圈資料
      MEP
      SET     M4160  ; [PPID]  配方搜尋KP
2151  LDD=    K0 D8720  ; SECS_上位傳PP_SEL-PPID
      ANDD=   K0 D8722  ; SECS_上位傳PP_SEL-PPID
      ANDD=   K0 D8724  ; SECS_上位傳PP_SEL-PPID
      ANDD=   K0 D8726  ; SECS_上位傳PP_SEL-PPID
      ANDD=   K0 D8728  ; SECS_上位傳PP_SEL-PPID
      INV
      OUT     M4150  ; [PPID]  判斷配方ID不為零-1
2173  LD=     H2020 D8720  ; SECS_上位傳PP_SEL-PPID
      AND=    H2020 D8721  ; SECS_上位傳PP_SEL-PPID
      AND=    H2020 D8722  ; SECS_上位傳PP_SEL-PPID
      AND=    H2020 D8723  ; SECS_上位傳PP_SEL-PPID
      AND=    H2020 D8724  ; SECS_上位傳PP_SEL-PPID
      AND=    H2020 D8725  ; SECS_上位傳PP_SEL-PPID
      AND=    H2020 D8726  ; SECS_上位傳PP_SEL-PPID
      AND=    H2020 D8727  ; SECS_上位傳PP_SEL-PPID
      AND=    H2020 D8728  ; SECS_上位傳PP_SEL-PPID
      AND=    H2020 D8729  ; SECS_上位傳PP_SEL-PPID
      INV
      OUT     M4151  ; [PPID]  判斷配判斷配方ID不為零-2
2205  LD      M4150  ; [PPID]  判斷配方ID不為零-1
      AND     M4151  ; [PPID]  判斷配判斷配方ID不為零-2
      OUT     M4152  ; [PPID]  判斷配方ID有效
2208  LD      SM400  ; PLC ON
      MOV     K0 Z14
      MOV     K0 Z15
      MOV     K0 Z8
2215  FOR     K30
2217  LD      M4160  ; [PPID]  配方搜尋KP
      AND     M4150  ; [PPID]  判斷配方ID不為零-1
      AND     M4151  ; [PPID]  判斷配判斷配方ID不為零-2
      ANDD=   D8720 ZR5300Z8  ; SECS_上位傳PP_SEL-PPID
      ANDD=   D8722 ZR5302Z8  ; SECS_上位傳PP_SEL-PPID
      AND=    D8724 ZR5304Z8  ; SECS_上位傳PP_SEL-PPID
      SET     M4161  ; [PPID]  配方搜尋比對OK
2233  LD      M4161  ; [PPID]  配方搜尋比對OK
      LD      M295  ; 配方切換旗標
      OR      SM400  ; PLC ON
      ANB
      MEP
      MOV     ZR10029Z14 D999  ; 生產呼叫SV
2241  LD<>    D0 K17  ; 人機現在畫頁
      AND     SM401
      MOVP    K1 D998  ; 溫度配方NO
2248  LDI     M6104  ; 回上位當前使用配方變更
      ANI     M4161  ; [PPID]  配方搜尋比對OK
      MOV     D999 D5520
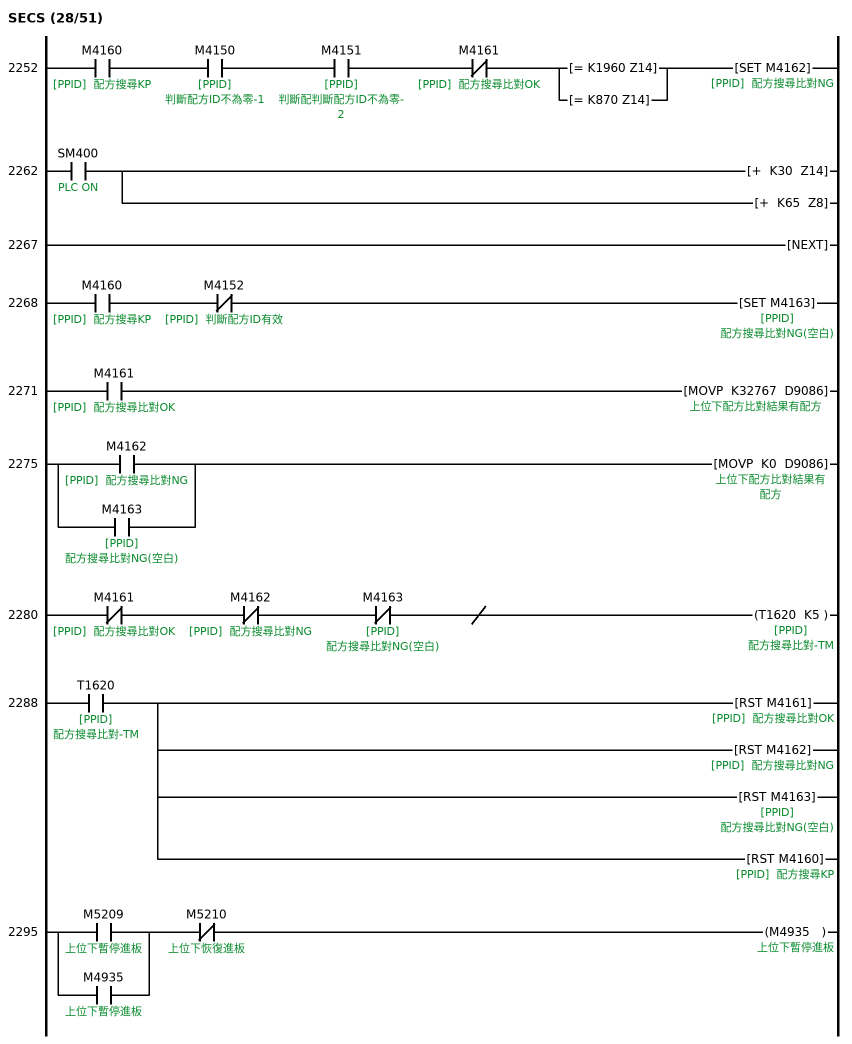
2252  LD      M4160  ; [PPID]  配方搜尋KP
      AND     M4150  ; [PPID]  判斷配方ID不為零-1
      AND     M4151  ; [PPID]  判斷配判斷配方ID不為零-2
      ANI     M4161  ; [PPID]  配方搜尋比對OK
      LD=     K1960 Z14
      OR=     K870 Z14
      ANB
      SET     M4162  ; [PPID]  配方搜尋比對NG
2262  LD      SM400  ; PLC ON
      +       K30 Z14
      +       K65 Z8
2267  NEXT
2268  LD      M4160  ; [PPID]  配方搜尋KP
      ANI     M4152  ; [PPID]  判斷配方ID有效
      SET     M4163  ; [PPID]  配方搜尋比對NG(空白)
2271  LD      M4161  ; [PPID]  配方搜尋比對OK
      MOVP    K32767 D9086
2275  LD      M4162  ; [PPID]  配方搜尋比對NG
      OR      M4163  ; [PPID]  配方搜尋比對NG(空白)
      MOVP    K0 D9086
2280  LDI     M4161  ; [PPID]  配方搜尋比對OK
      ANI     M4162  ; [PPID]  配方搜尋比對NG
      ANI     M4163  ; [PPID]  配方搜尋比對NG(空白)
      INV
      OUT     T1620 K5  ; [PPID]  配方搜尋比對-TM
2288  LD      T1620  ; [PPID]  配方搜尋比對-TM
      RST     M4161  ; [PPID]  配方搜尋比對OK
      RST     M4162  ; [PPID]  配方搜尋比對NG
      RST     M4163  ; [PPID]  配方搜尋比對NG(空白)
      RST     M4160  ; [PPID]  配方搜尋KP
2295  LD      M5209  ; 上位下暫停進板
      OR      M4935  ; 上位下暫停進板
      ANI     M5210  ; 上位下恢復進板
      OUT     M4935  ; 上位下暫停進板
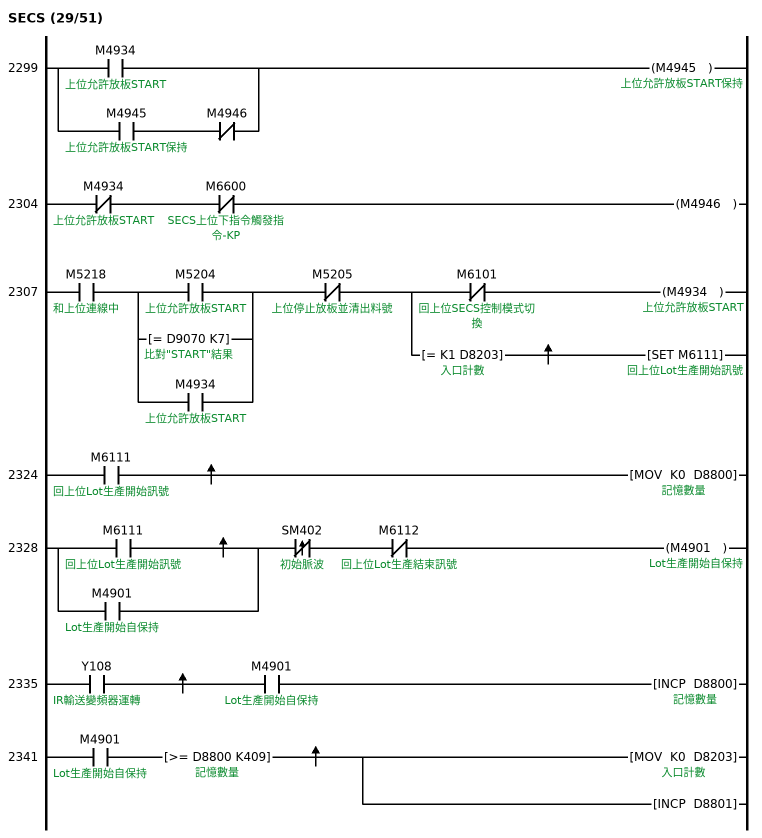
2299  LD      M4934  ; 上位允許放板START
      LD      M4945  ; 上位允許放板START保持
      ANI     M4946
      ORB
      OUT     M4945  ; 上位允許放板START保持
2304  LDI     M4934  ; 上位允許放板START
      ANI     M6600  ; SECS上位下指令觸發指令-KP
      OUT     M4946
2307  LD      M5218  ; 和上位連線中
      LD      M5204  ; 上位允許放板START
      OR=     D9070 K7  ; 比對"START"結果
      OR      M4934  ; 上位允許放板START
      ANB
      ANI     M5205  ; 上位停止放板並清出料號
      MPS
      ANI     M6101  ; 回上位SECS控制模式切換
      OUT     M4934  ; 上位允許放板START
      MPP
      AND=    K1 D8203  ; 入口計數
      MEP
      SET     M6111  ; 回上位Lot生產開始訊號
2324  LD      M6111  ; 回上位Lot生產開始訊號
      MEP
      MOV     K0 D8800  ; 記憶數量
2328  LD      M6111  ; 回上位Lot生產開始訊號
      MEP
      OR      M4901  ; Lot生產開始自保持
      ANDPI   SM402  ; 初始脈波
      ANI     M6112  ; 回上位Lot生產結束訊號
      OUT     M4901  ; Lot生產開始自保持
2335  LD      Y108  ; IR輸送變頻器運轉
      MEP
      AND     M4901  ; Lot生產開始自保持
      INCP    D8800
2341  LD      M4901  ; Lot生產開始自保持
      AND>=   D8800 K409  ; 記憶數量
      MEP
      MOV     K0 D8203
      INCP    D8801
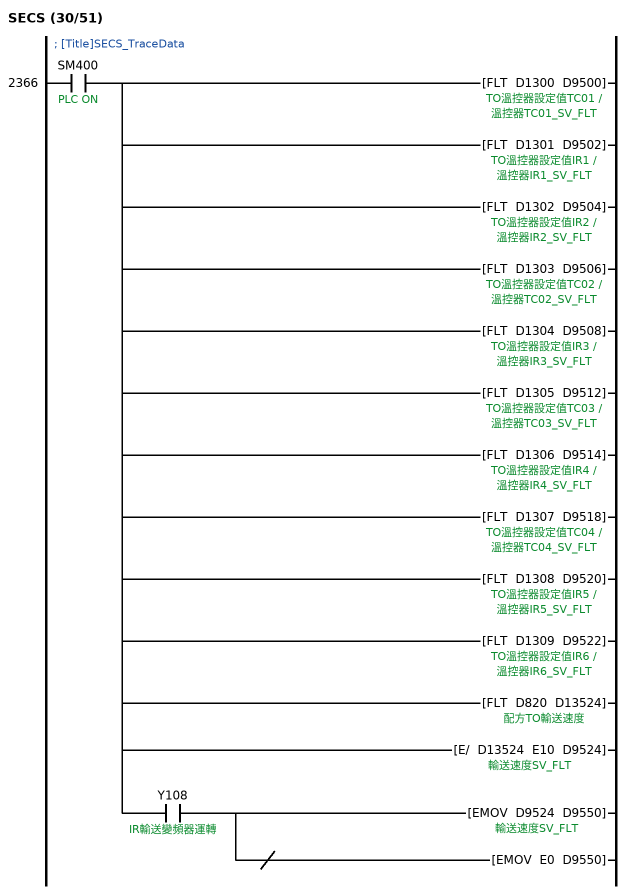
; [Title]SECS_TraceData
2366  LD      SM400  ; PLC ON
      FLT     D1300 D9500  ; TO溫控器設定值TC01 / 溫控器TC01_SV_FLT
      FLT     D1301 D9502  ; TO溫控器設定值IR1 / 溫控器IR1_SV_FLT
      FLT     D1302 D9504  ; TO溫控器設定值IR2 / 溫控器IR2_SV_FLT
      FLT     D1303 D9506  ; TO溫控器設定值TC02 / 溫控器TC02_SV_FLT
      FLT     D1304 D9508  ; TO溫控器設定值IR3 / 溫控器IR3_SV_FLT
      FLT     D1305 D9512  ; TO溫控器設定值TC03 / 溫控器TC03_SV_FLT
      FLT     D1306 D9514  ; TO溫控器設定值IR4 / 溫控器IR4_SV_FLT
      FLT     D1307 D9518  ; TO溫控器設定值TC04 / 溫控器TC04_SV_FLT
      FLT     D1308 D9520  ; TO溫控器設定值IR5 / 溫控器IR5_SV_FLT
      FLT     D1309 D9522  ; TO溫控器設定值IR6 / 溫控器IR6_SV_FLT
      FLT     D820 D13524  ; 配方TO輸送速度
      E/      D13524 E10 D9524  ; 輸送速度SV_FLT
      AND     Y108  ; IR輸送變頻器運轉
      EMOV    D9524 D9550
      INV
      EMOV    E0 D9550
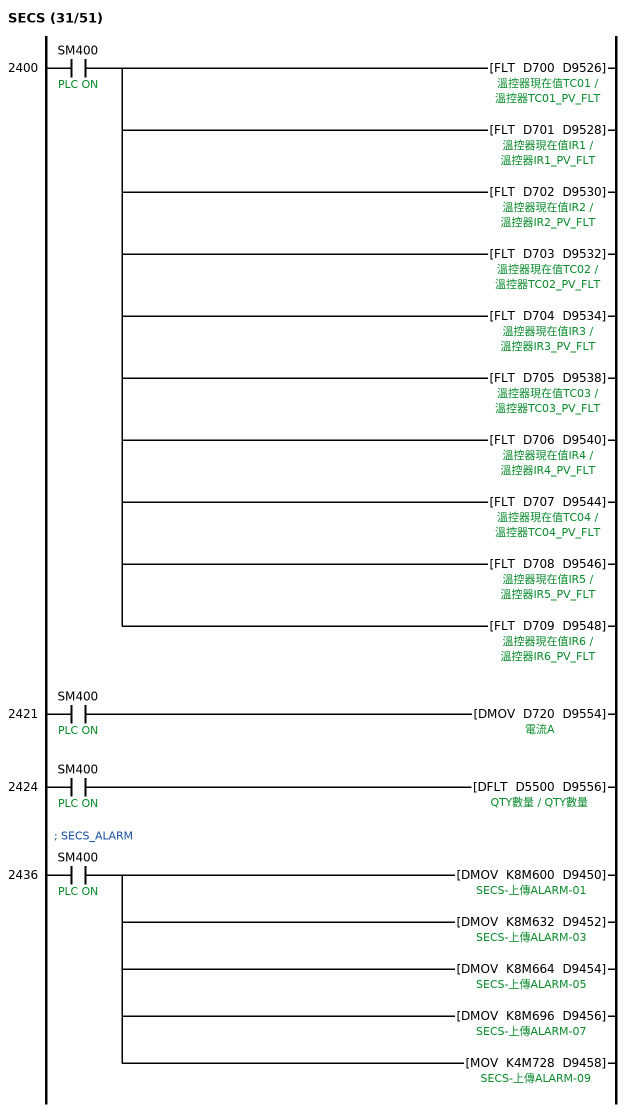
2400  LD      SM400  ; PLC ON
      FLT     D700 D9526  ; 溫控器現在值TC01 / 溫控器TC01_PV_FLT
      FLT     D701 D9528  ; 溫控器現在值IR1 / 溫控器IR1_PV_FLT
      FLT     D702 D9530  ; 溫控器現在值IR2 / 溫控器IR2_PV_FLT
      FLT     D703 D9532  ; 溫控器現在值TC02 / 溫控器TC02_PV_FLT
      FLT     D704 D9534  ; 溫控器現在值IR3 / 溫控器IR3_PV_FLT
      FLT     D705 D9538  ; 溫控器現在值TC03 / 溫控器TC03_PV_FLT
      FLT     D706 D9540  ; 溫控器現在值IR4 / 溫控器IR4_PV_FLT
      FLT     D707 D9544  ; 溫控器現在值TC04 / 溫控器TC04_PV_FLT
      FLT     D708 D9546  ; 溫控器現在值IR5 / 溫控器IR5_PV_FLT
      FLT     D709 D9548  ; 溫控器現在值IR6 / 溫控器IR6_PV_FLT
2421  LD      SM400  ; PLC ON
      DMOV    D720 D9554  ; 電流A
2424  LD      SM400  ; PLC ON
      DFLT    D5500 D9556  ; QTY數量
; SECS_ALARM
2436  LD      SM400  ; PLC ON
      DMOV    K8M600 D9450  ; 緊急停止 / SECS-上傳ALARM-01
      DMOV    K8M632 D9452  ; 第十三槽電熱超溫異常 / SECS-上傳ALARM-03
      DMOV    K8M664 D9454  ; SECS-上傳ALARM-05
      DMOV    K8M696 D9456  ; 第二槽IR3超溫防止器異常 / SECS-上傳ALARM-07
      MOV     K4M728 D9458  ; 第十一槽SCR異常 / SECS-上傳ALARM-09
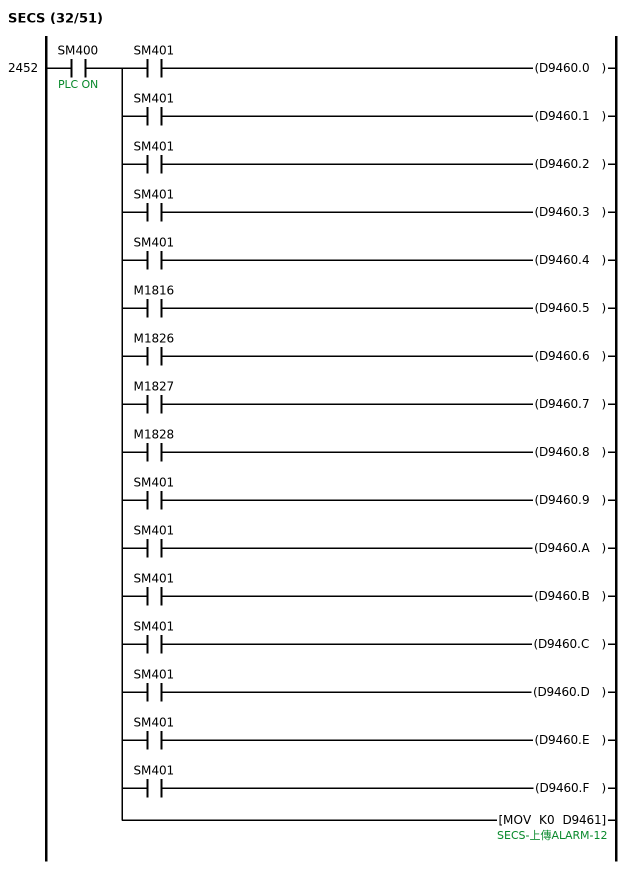
2452  LD      SM400  ; PLC ON
      MPS
      AND     SM401
      OUT     D9460.0
      MRD
      AND     SM401
      OUT     D9460.1
      MRD
      AND     SM401
      OUT     D9460.2
      MRD
      AND     SM401
      OUT     D9460.3
      MRD
      AND     SM401
      OUT     D9460.4
      MRD
      AND     M1816
      OUT     D9460.5
      MRD
      AND     M1826
      OUT     D9460.6
      MRD
      AND     M1827
      OUT     D9460.7
      MRD
      AND     M1828
      OUT     D9460.8
      MRD
      AND     SM401
      OUT     D9460.9
      MRD
      AND     SM401
      OUT     D9460.A
      MRD
      AND     SM401
      OUT     D9460.B
      MRD
      AND     SM401
      OUT     D9460.C
      MRD
      AND     SM401
      OUT     D9460.D
      MRD
      AND     SM401
      OUT     D9460.E
      MRD
      AND     SM401
      OUT     D9460.F
      MPP
      MOV     K0 D9461  ; SECS-上傳ALARM-12
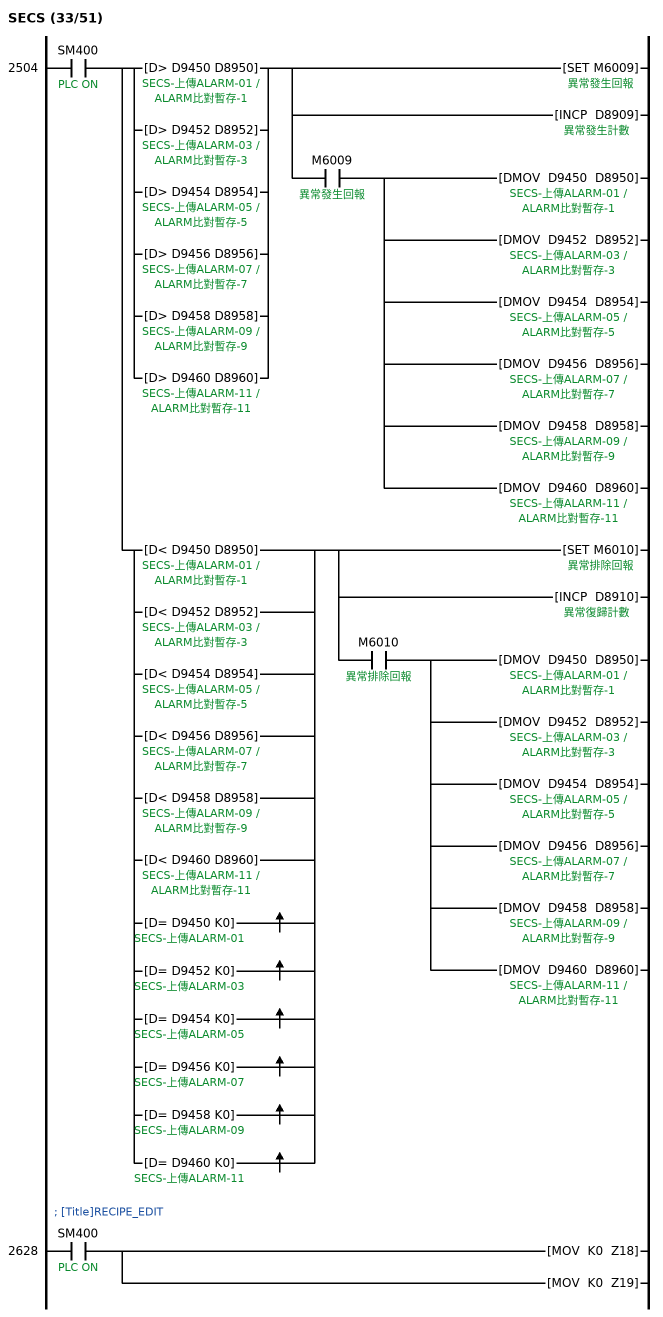
2504  LD      SM400  ; PLC ON
      MPS
      LDD>    D9450 D8950  ; SECS-上傳ALARM-01 / ALARM比對暫存-1
      ORD>    D9452 D8952  ; SECS-上傳ALARM-03 / ALARM比對暫存-3
      ORD>    D9454 D8954  ; SECS-上傳ALARM-05 / ALARM比對暫存-5
      ORD>    D9456 D8956  ; SECS-上傳ALARM-07 / ALARM比對暫存-7
      ORD>    D9458 D8958  ; SECS-上傳ALARM-09 / ALARM比對暫存-9
      ORD>    D9460 D8960  ; SECS-上傳ALARM-11 / ALARM比對暫存-11
      ANB
      SET     M6009  ; 異常發生回報
      INCP    D8909  ; 異常發生計數
      AND     M6009  ; 異常發生回報
      DMOV    D9450 D8950
      DMOV    D9452 D8952
      DMOV    D9454 D8954
      DMOV    D9456 D8956
      DMOV    D9458 D8958
      DMOV    D9460 D8960
      MPP
      LDD<    D9450 D8950  ; SECS-上傳ALARM-01 / ALARM比對暫存-1
      ORD<    D9452 D8952  ; SECS-上傳ALARM-03 / ALARM比對暫存-3
      ORD<    D9454 D8954  ; SECS-上傳ALARM-05 / ALARM比對暫存-5
      ORD<    D9456 D8956  ; SECS-上傳ALARM-07 / ALARM比對暫存-7
      ORD<    D9458 D8958  ; SECS-上傳ALARM-09 / ALARM比對暫存-9
      ORD<    D9460 D8960  ; SECS-上傳ALARM-11 / ALARM比對暫存-11
      LDD=    D9450 K0  ; SECS-上傳ALARM-01
      MEP
      ORB
      LDD=    D9452 K0  ; SECS-上傳ALARM-03
      MEP
      ORB
      LDD=    D9454 K0  ; SECS-上傳ALARM-05
      MEP
      ORB
      LDD=    D9456 K0  ; SECS-上傳ALARM-07
      MEP
      ORB
      LDD=    D9458 K0  ; SECS-上傳ALARM-09
      MEP
      ORB
      LDD=    D9460 K0  ; SECS-上傳ALARM-11
      MEP
      ORB
      ANB
      SET     M6010  ; 異常排除回報
      INCP    D8910  ; 異常復歸計數
      AND     M6010  ; 異常排除回報
      DMOV    D9450 D8950
      DMOV    D9452 D8952
      DMOV    D9454 D8954
      DMOV    D9456 D8956
      DMOV    D9458 D8958
      DMOV    D9460 D8960
; [Title]RECIPE_EDIT
2628  LD      SM400  ; PLC ON
      MOV     K0 Z18
      MOV     K0 Z19
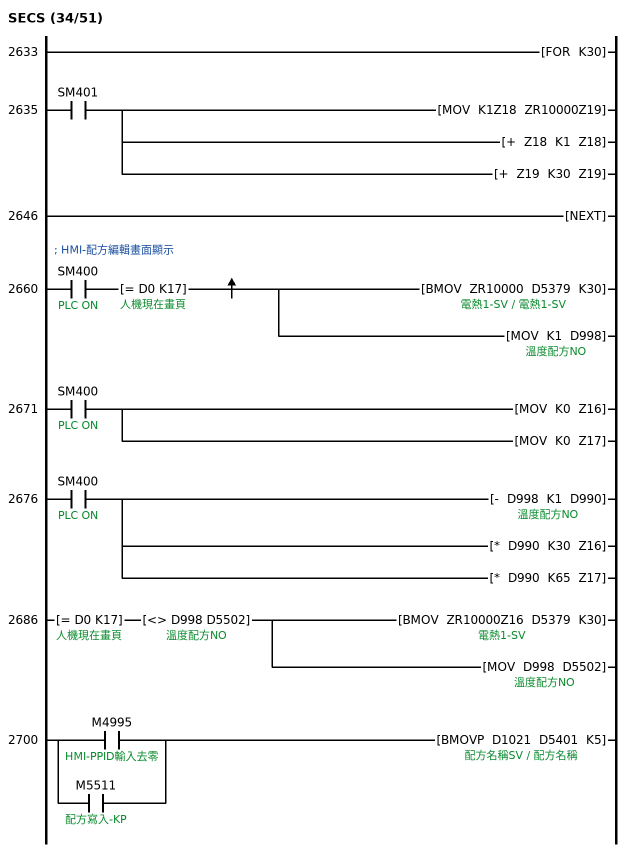
2633  FOR     K30
2635  LD      SM401
      MOV     K1Z18 ZR10000Z19
      +       Z18 K1 Z18
      +       Z19 K30 Z19
2646  NEXT
; HMI-配方編輯畫面顯示
2660  LD      SM400  ; PLC ON
      AND=    D0 K17  ; 人機現在畫頁
      MEP
      BMOV    ZR10000 D5379 K30  ; 電熱1-SV / 電熱1-SV
      MOV     K1 D998
2671  LD      SM400  ; PLC ON
      MOV     K0 Z16
      MOV     K0 Z17
2676  LD      SM400  ; PLC ON
      -       D998 K1 D990
      *       D990 K30 Z16
      *       D990 K65 Z17
2686  LD=     D0 K17  ; 人機現在畫頁
      AND<>   D998 D5502  ; 溫度配方NO
      BMOV    ZR10000Z16 D5379 K30
      MOV     D998 D5502
2700  LD      M4995  ; HMI-PPID輸入去零
      OR      M5511  ; 配方寫入-KP
      BMOVP   D1021 D5401 K5  ; 配方名稱SV / 配方名稱
